RoboDK station: path.rdk

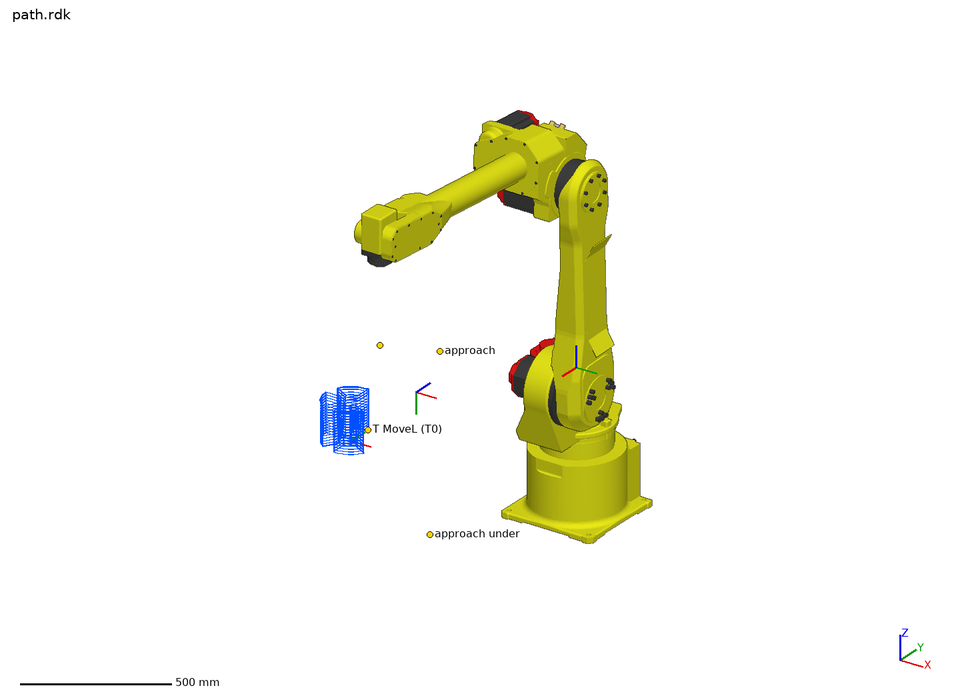
[picture v0: the station drawn from its stored meshes, robots at their saved joint values, targets as dots, program paths as lines]
Station path (saved by RoboDK 5.0.0). Poses are relative to the parent item; angles as X-Y-Z fixed-axis rotations.
  - frame data_frame at (0, 0, 0) mm
    - target approach (Cartesian target) at (94, 380, 204.2) mm, rotated rx -180 ry 0 rz 0 deg; joints [10.247, -49.52, -8.659, -50.211, 13.385, 139.433] of Fanuc ARC Mate 120iB/10L
    - target approach_vert (Cartesian target) at (0, 170, 284.2) mm, rotated rx -90 ry 0 rz 180 deg; joints [0, 2.156, 3.881, -180, 93.881, 90] of Fanuc ARC Mate 120iB/10L
    - target approach under (Cartesian target) at (94, 320, -445.8) mm; joints [3.897, 48.417, -53.03, 175.127, 126.871, 267.072] of Fanuc ARC Mate 120iB/10L
    - target approach_vert_180 (Cartesian target) at (0, 170, 284.2) mm, rotated rx -90 ry 0 rz 0 deg; joints [0, 2.156, 3.881, -180, 93.881, -90] of Fanuc ARC Mate 120iB/10L
    - object path at (0, 0, 0) mm
    - target T MoveL (T0) (Cartesian target) at (0, 100, 0) mm, rotated rx -90 ry 0 rz 0 deg; joints [0, 0, 0, 0, 0, 0] of Fanuc ARC Mate 120iB/10L
  - frame Fanuc ARC Mate 120iB/10L Base at (0, 1300, -250) mm, rotated rx 0 ry 0 rz -90 deg
    - robot Fanuc ARC Mate 120iB/10L: 6 axes, payload 10 kg, reach 1885 mm, repeatability 0.1 mm, weight 225 kg
        modified DH rows (alpha deg, a mm, theta deg, d mm): 0, 0, 0, 525; -90, 150, -90, 0; 0, 770, 0, 0; -90, 100, 0, 960; 90, 0, 0, 0; -90, 0, 0, 100
        base shift (0, 0, -525) mm
        joint limits [-170, -80, -170, -200, -140, -450] to [170, 170, 250, 200, 140, 450]; home [0, 0, 0, 0, 0, 0]; saved at [0, 2.156, 3.881, -180, 93.881, -90]
      - tool Tool 1, TCP at (0, 0, 300) mm, rotated rx 90 ry 0 rz 0 deg
      - tool Tool 2, TCP at (0, 0, 200) mm
      - tool Tool 3, TCP at (0, 0, 300) mm, rotated rx -90 ry 0 rz 0 deg
  - frame Frame 3 at (130, 190, 140) mm, rotated rx -90 ry 0 rz 0 deg
  - program AutoProgram (841 instructions, listed below)
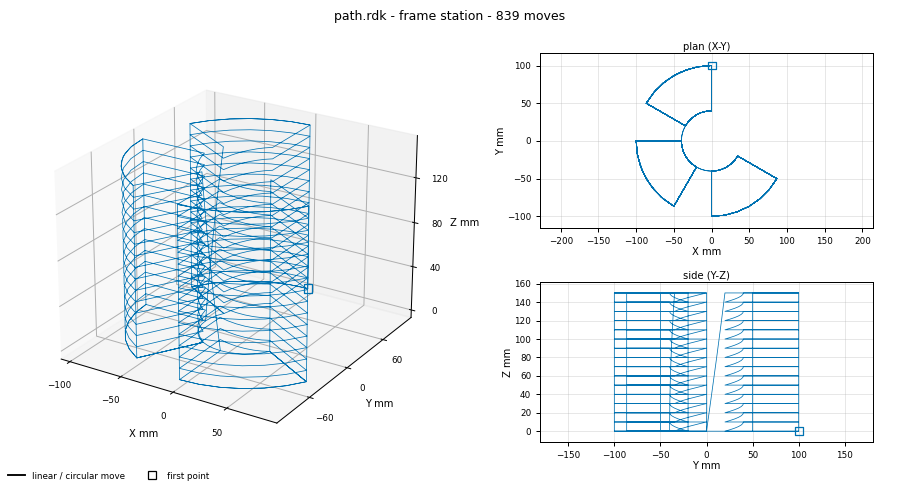
[picture p0: tool path of path.rdk in frame station, 839 of 839 moves have a stored position in this frame; points joined in program order, loops and branches not executed]

--- program AutoProgram (robot Fanuc ARC Mate 120iB/10L) ---
  Set Ref.: data_frame
  Set Tool: Tool 1
  *MoveL (T0) -> target T MoveL (T0)
  MoveL (T1) to (-17.36, 98.48, 0) mm, rotated rx -90 ry 0 rz 10 deg; joints []
  MoveL (T2) to (-34.2, 93.97, 0) mm, rotated rx -90 ry 0 rz 20 deg; joints []
  MoveL (T3) to (-50, 86.6, 0) mm, rotated rx -90 ry 0 rz 30 deg; joints []
  MoveL (T4) to (-64.28, 76.6, 0) mm, rotated rx -90 ry 0 rz 40 deg; joints []
  MoveL (T5) to (-76.6, 64.28, 0) mm, rotated rx -90 ry 0 rz 50 deg; joints []
  MoveL (T6) to (-86.6, 50, 0) mm, rotated rx -90 ry 0 rz 60 deg; joints []
  MoveL (T7) to (-34.64, 20, 0) mm, rotated rx -90 ry 0 rz 60 deg; joints []
  MoveL (T8) to (-30.64, 25.71, 1.67) mm, rotated rx -90 ry 0 rz 50 deg; joints []
  MoveL (T9) to (-25.71, 30.64, 3.33) mm, rotated rx -90 ry 0 rz 40 deg; joints []
  MoveL (T10) to (-20, 34.64, 5) mm, rotated rx -90 ry 0 rz 30 deg; joints []
  MoveL (T11) to (-13.68, 37.59, 6.67) mm, rotated rx -90 ry 0 rz 20 deg; joints []
  MoveL (T12) to (-6.95, 39.39, 8.33) mm, rotated rx -90 ry 0 rz 10 deg; joints []
  MoveL (T13) to (0, 40, 10) mm, rotated rx -90 ry 0 rz 0 deg; joints []
  MoveL (T14) to (0, 100, 10) mm, rotated rx -90 ry 0 rz 0 deg; joints []
  MoveL (T15) to (-17.36, 98.48, 10) mm, rotated rx -90 ry 0 rz 10 deg; joints []
  MoveL (T16) to (-34.2, 93.97, 10) mm, rotated rx -90 ry 0 rz 20 deg; joints []
  MoveL (T17) to (-50, 86.6, 10) mm, rotated rx -90 ry 0 rz 30 deg; joints []
  MoveL (T18) to (-64.28, 76.6, 10) mm, rotated rx -90 ry 0 rz 40 deg; joints []
  MoveL (T19) to (-76.6, 64.28, 10) mm, rotated rx -90 ry 0 rz 50 deg; joints []
  MoveL (T20) to (-86.6, 50, 10) mm, rotated rx -90 ry 0 rz 60 deg; joints []
  MoveL (T21) to (-34.64, 20, 10) mm, rotated rx -90 ry 0 rz 60 deg; joints []
  MoveL (T22) to (-30.64, 25.71, 11.67) mm, rotated rx -90 ry 0 rz 50 deg; joints []
  MoveL (T23) to (-25.71, 30.64, 13.33) mm, rotated rx -90 ry 0 rz 40 deg; joints []
  MoveL (T24) to (-20, 34.64, 15) mm, rotated rx -90 ry 0 rz 30 deg; joints []
  MoveL (T25) to (-13.68, 37.59, 16.67) mm, rotated rx -90 ry 0 rz 20 deg; joints []
  MoveL (T26) to (-6.95, 39.39, 18.33) mm, rotated rx -90 ry 0 rz 10 deg; joints []
  MoveL (T27) to (0, 40, 20) mm, rotated rx -90 ry 0 rz 0 deg; joints []
  MoveL (T28) to (0, 100, 20) mm, rotated rx -90 ry 0 rz 0 deg; joints []
  MoveL (T29) to (-17.36, 98.48, 20) mm, rotated rx -90 ry 0 rz 10 deg; joints []
  MoveL (T30) to (-34.2, 93.97, 20) mm, rotated rx -90 ry 0 rz 20 deg; joints []
  MoveL (T31) to (-50, 86.6, 20) mm, rotated rx -90 ry 0 rz 30 deg; joints []
  MoveL (T32) to (-64.28, 76.6, 20) mm, rotated rx -90 ry 0 rz 40 deg; joints []
  MoveL (T33) to (-76.6, 64.28, 20) mm, rotated rx -90 ry 0 rz 50 deg; joints []
  MoveL (T34) to (-86.6, 50, 20) mm, rotated rx -90 ry 0 rz 60 deg; joints []
  MoveL (T35) to (-34.64, 20, 20) mm, rotated rx -90 ry 0 rz 60 deg; joints []
  MoveL (T36) to (-30.64, 25.71, 21.67) mm, rotated rx -90 ry 0 rz 50 deg; joints []
  MoveL (T37) to (-25.71, 30.64, 23.33) mm, rotated rx -90 ry 0 rz 40 deg; joints []
  MoveL (T38) to (-20, 34.64, 25) mm, rotated rx -90 ry 0 rz 30 deg; joints []
  MoveL (T39) to (-13.68, 37.59, 26.67) mm, rotated rx -90 ry 0 rz 20 deg; joints []
  MoveL (T40) to (-6.95, 39.39, 28.33) mm, rotated rx -90 ry 0 rz 10 deg; joints []
  MoveL (T41) to (0, 40, 30) mm, rotated rx -90 ry 0 rz 0 deg; joints []
  MoveL (T42) to (0, 100, 30) mm, rotated rx -90 ry 0 rz 0 deg; joints []
  MoveL (T43) to (-20.79, 97.81, 30) mm, rotated rx -90 ry 0 rz 12 deg; joints []
  MoveL (T44) to (-40.67, 91.36, 30) mm, rotated rx -90 ry 0 rz 24 deg; joints []
  MoveL (T45) to (-58.78, 80.9, 30) mm, rotated rx -90 ry 0 rz 36 deg; joints []
  MoveL (T46) to (-74.31, 66.91, 30) mm, rotated rx -90 ry 0 rz 48 deg; joints []
  MoveL (T47) to (-86.6, 50, 30) mm, rotated rx -90 ry 0 rz 60 deg; joints []
  MoveL (T48) to (-34.64, 20, 30) mm, rotated rx -90 ry 0 rz 60 deg; joints []
  MoveL (T49) to (-30.64, 25.71, 31.67) mm, rotated rx -90 ry 0 rz 50 deg; joints []
  MoveL (T50) to (-25.71, 30.64, 33.33) mm, rotated rx -90 ry 0 rz 40 deg; joints []
  MoveL (T51) to (-20, 34.64, 35) mm, rotated rx -90 ry 0 rz 30 deg; joints []
  MoveL (T52) to (-13.68, 37.59, 36.67) mm, rotated rx -90 ry 0 rz 20 deg; joints []
  MoveL (T53) to (-6.95, 39.39, 38.33) mm, rotated rx -90 ry 0 rz 10 deg; joints []
  MoveL (T54) to (0, 40, 40) mm, rotated rx -90 ry 0 rz 0 deg; joints []
  MoveL (T55) to (0, 100, 40) mm, rotated rx -90 ry 0 rz 0 deg; joints []
  MoveL (T56) to (-17.36, 98.48, 40) mm, rotated rx -90 ry 0 rz 10 deg; joints []
  MoveL (T57) to (-34.2, 93.97, 40) mm, rotated rx -90 ry 0 rz 20 deg; joints []
  MoveL (T58) to (-50, 86.6, 40) mm, rotated rx -90 ry 0 rz 30 deg; joints []
  MoveL (T59) to (-64.28, 76.6, 40) mm, rotated rx -90 ry 0 rz 40 deg; joints []
  MoveL (T60) to (-76.6, 64.28, 40) mm, rotated rx -90 ry 0 rz 50 deg; joints []
  MoveL (T61) to (-86.6, 50, 40) mm, rotated rx -90 ry 0 rz 60 deg; joints []
  MoveL (T62) to (-34.64, 20, 40) mm, rotated rx -90 ry 0 rz 60 deg; joints []
  MoveL (T63) to (-30.64, 25.71, 41.67) mm, rotated rx -90 ry 0 rz 50 deg; joints []
  MoveL (T64) to (-25.71, 30.64, 43.33) mm, rotated rx -90 ry 0 rz 40 deg; joints []
  MoveL (T65) to (-20, 34.64, 45) mm, rotated rx -90 ry 0 rz 30 deg; joints []
  MoveL (T66) to (-13.68, 37.59, 46.67) mm, rotated rx -90 ry 0 rz 20 deg; joints []
  MoveL (T67) to (-6.95, 39.39, 48.33) mm, rotated rx -90 ry 0 rz 10 deg; joints []
  MoveL (T68) to (0, 40, 50) mm, rotated rx -90 ry 0 rz 0 deg; joints []
  MoveL (T69) to (0, 100, 50) mm, rotated rx -90 ry 0 rz 0 deg; joints []
  MoveL (T70) to (-17.36, 98.48, 50) mm, rotated rx -90 ry 0 rz 10 deg; joints []
  MoveL (T71) to (-34.2, 93.97, 50) mm, rotated rx -90 ry 0 rz 20 deg; joints []
  MoveL (T72) to (-50, 86.6, 50) mm, rotated rx -90 ry 0 rz 30 deg; joints []
  MoveL (T73) to (-64.28, 76.6, 50) mm, rotated rx -90 ry 0 rz 40 deg; joints []
  MoveL (T74) to (-76.6, 64.28, 50) mm, rotated rx -90 ry 0 rz 50 deg; joints []
  MoveL (T75) to (-86.6, 50, 50) mm, rotated rx -90 ry 0 rz 60 deg; joints []
  MoveL (T76) to (-34.64, 20, 50) mm, rotated rx -90 ry 0 rz 60 deg; joints []
  MoveL (T77) to (-30.64, 25.71, 51.67) mm, rotated rx -90 ry 0 rz 50 deg; joints []
  MoveL (T78) to (-25.71, 30.64, 53.33) mm, rotated rx -90 ry 0 rz 40 deg; joints []
  MoveL (T79) to (-20, 34.64, 55) mm, rotated rx -90 ry 0 rz 30 deg; joints []
  MoveL (T80) to (-13.68, 37.59, 56.67) mm, rotated rx -90 ry 0 rz 20 deg; joints []
  MoveL (T81) to (-6.95, 39.39, 58.33) mm, rotated rx -90 ry 0 rz 10 deg; joints []
  MoveL (T82) to (0, 40, 60) mm, rotated rx -90 ry 0 rz 0 deg; joints []
  MoveL (T83) to (0, 100, 60) mm, rotated rx -90 ry 0 rz 0 deg; joints []
  MoveL (T84) to (-17.36, 98.48, 60) mm, rotated rx -90 ry 0 rz 10 deg; joints []
  MoveL (T85) to (-34.2, 93.97, 60) mm, rotated rx -90 ry 0 rz 20 deg; joints []
  MoveL (T86) to (-50, 86.6, 60) mm, rotated rx -90 ry 0 rz 30 deg; joints []
  MoveL (T87) to (-64.28, 76.6, 60) mm, rotated rx -90 ry 0 rz 40 deg; joints []
  MoveL (T88) to (-76.6, 64.28, 60) mm, rotated rx -90 ry 0 rz 50 deg; joints []
  MoveL (T89) to (-86.6, 50, 60) mm, rotated rx -90 ry 0 rz 60 deg; joints []
  MoveL (T90) to (-34.64, 20, 60) mm, rotated rx -90 ry 0 rz 60 deg; joints []
  MoveL (T91) to (-30.64, 25.71, 61.67) mm, rotated rx -90 ry 0 rz 50 deg; joints []
  MoveL (T92) to (-25.71, 30.64, 63.33) mm, rotated rx -90 ry 0 rz 40 deg; joints []
  MoveL (T93) to (-20, 34.64, 65) mm, rotated rx -90 ry 0 rz 30 deg; joints []
  MoveL (T94) to (-13.68, 37.59, 66.67) mm, rotated rx -90 ry 0 rz 20 deg; joints []
  MoveL (T95) to (-6.95, 39.39, 68.33) mm, rotated rx -90 ry 0 rz 10 deg; joints []
  MoveL (T96) to (0, 40, 70) mm, rotated rx -90 ry 0 rz 0 deg; joints []
  MoveL (T97) to (0, 100, 70) mm, rotated rx -90 ry 0 rz 0 deg; joints []
  MoveL (T98) to (-17.36, 98.48, 70) mm, rotated rx -90 ry 0 rz 10 deg; joints []
  MoveL (T99) to (-34.2, 93.97, 70) mm, rotated rx -90 ry 0 rz 20 deg; joints []
  MoveL (T100) to (-50, 86.6, 70) mm, rotated rx -90 ry 0 rz 30 deg; joints []
  MoveL (T101) to (-64.28, 76.6, 70) mm, rotated rx -90 ry 0 rz 40 deg; joints []
  MoveL (T102) to (-76.6, 64.28, 70) mm, rotated rx -90 ry 0 rz 50 deg; joints []
  MoveL (T103) to (-86.6, 50, 70) mm, rotated rx -90 ry 0 rz 60 deg; joints []
  MoveL (T104) to (-34.64, 20, 70) mm, rotated rx -90 ry 0 rz 60 deg; joints []
  MoveL (T105) to (-30.64, 25.71, 71.67) mm, rotated rx -90 ry 0 rz 50 deg; joints []
  MoveL (T106) to (-25.71, 30.64, 73.33) mm, rotated rx -90 ry 0 rz 40 deg; joints []
  MoveL (T107) to (-20, 34.64, 75) mm, rotated rx -90 ry 0 rz 30 deg; joints []
  MoveL (T108) to (-13.68, 37.59, 76.67) mm, rotated rx -90 ry 0 rz 20 deg; joints []
  MoveL (T109) to (-6.95, 39.39, 78.33) mm, rotated rx -90 ry 0 rz 10 deg; joints []
  MoveL (T110) to (0, 40, 80) mm, rotated rx -90 ry 0 rz 0 deg; joints []
  MoveL (T111) to (0, 100, 80) mm, rotated rx -90 ry 0 rz 0 deg; joints []
  MoveL (T112) to (-20.79, 97.81, 80) mm, rotated rx -90 ry 0 rz 12 deg; joints []
  MoveL (T113) to (-40.67, 91.36, 80) mm, rotated rx -90 ry 0 rz 24 deg; joints []
  MoveL (T114) to (-58.78, 80.9, 80) mm, rotated rx -90 ry 0 rz 36 deg; joints []
  MoveL (T115) to (-74.31, 66.91, 80) mm, rotated rx -90 ry 0 rz 48 deg; joints []
  MoveL (T116) to (-86.6, 50, 80) mm, rotated rx -90 ry 0 rz 60 deg; joints []
  MoveL (T117) to (-34.64, 20, 80) mm, rotated rx -90 ry 0 rz 60 deg; joints []
  MoveL (T118) to (-30.64, 25.71, 81.67) mm, rotated rx -90 ry 0 rz 50 deg; joints []
  MoveL (T119) to (-25.71, 30.64, 83.33) mm, rotated rx -90 ry 0 rz 40 deg; joints []
  MoveL (T120) to (-20, 34.64, 85) mm, rotated rx -90 ry 0 rz 30 deg; joints []
  MoveL (T121) to (-13.68, 37.59, 86.67) mm, rotated rx -90 ry 0 rz 20 deg; joints []
  MoveL (T122) to (-6.95, 39.39, 88.33) mm, rotated rx -90 ry 0 rz 10 deg; joints []
  MoveL (T123) to (0, 40, 90) mm, rotated rx -90 ry 0 rz 0 deg; joints []
  MoveL (T124) to (0, 100, 90) mm, rotated rx -90 ry 0 rz 0 deg; joints []
  MoveL (T125) to (-20.79, 97.81, 90) mm, rotated rx -90 ry 0 rz 12 deg; joints []
  MoveL (T126) to (-40.67, 91.36, 90) mm, rotated rx -90 ry 0 rz 24 deg; joints []
  MoveL (T127) to (-58.78, 80.9, 90) mm, rotated rx -90 ry 0 rz 36 deg; joints []
  MoveL (T128) to (-74.31, 66.91, 90) mm, rotated rx -90 ry 0 rz 48 deg; joints []
  MoveL (T129) to (-86.6, 50, 90) mm, rotated rx -90 ry 0 rz 60 deg; joints []
  MoveL (T130) to (-34.64, 20, 90) mm, rotated rx -90 ry 0 rz 60 deg; joints []
  MoveL (T131) to (-30.64, 25.71, 91.67) mm, rotated rx -90 ry 0 rz 50 deg; joints []
  MoveL (T132) to (-25.71, 30.64, 93.33) mm, rotated rx -90 ry 0 rz 40 deg; joints []
  MoveL (T133) to (-20, 34.64, 95) mm, rotated rx -90 ry 0 rz 30 deg; joints []
  MoveL (T134) to (-13.68, 37.59, 96.67) mm, rotated rx -90 ry 0 rz 20 deg; joints []
  MoveL (T135) to (-6.95, 39.39, 98.33) mm, rotated rx -90 ry 0 rz 10 deg; joints []
  MoveL (T136) to (0, 40, 100) mm, rotated rx -90 ry 0 rz 0 deg; joints []
  MoveL (T137) to (0, 100, 100) mm, rotated rx -90 ry 0 rz 0 deg; joints []
  MoveL (T138) to (-20.79, 97.81, 100) mm, rotated rx -90 ry 0 rz 12 deg; joints []
  MoveL (T139) to (-40.67, 91.36, 100) mm, rotated rx -90 ry 0 rz 24 deg; joints []
  MoveL (T140) to (-58.78, 80.9, 100) mm, rotated rx -90 ry 0 rz 36 deg; joints []
  MoveL (T141) to (-74.31, 66.91, 100) mm, rotated rx -90 ry 0 rz 48 deg; joints []
  MoveL (T142) to (-86.6, 50, 100) mm, rotated rx -90 ry 0 rz 60 deg; joints []
  MoveL (T143) to (-34.64, 20, 100) mm, rotated rx -90 ry 0 rz 60 deg; joints []
  MoveL (T144) to (-30.64, 25.71, 101.67) mm, rotated rx -90 ry 0 rz 50 deg; joints []
  MoveL (T145) to (-25.71, 30.64, 103.33) mm, rotated rx -90 ry 0 rz 40 deg; joints []
  MoveL (T146) to (-20, 34.64, 105) mm, rotated rx -90 ry 0 rz 30 deg; joints []
  MoveL (T147) to (-13.68, 37.59, 106.67) mm, rotated rx -90 ry 0 rz 20 deg; joints []
  MoveL (T148) to (-6.95, 39.39, 108.33) mm, rotated rx -90 ry 0 rz 10 deg; joints []
  MoveL (T149) to (0, 40, 110) mm, rotated rx -90 ry 0 rz 0 deg; joints []
  MoveL (T150) to (0, 100, 110) mm, rotated rx -90 ry 0 rz 0 deg; joints []
  MoveL (T151) to (-17.36, 98.48, 110) mm, rotated rx -90 ry 0 rz 10 deg; joints []
  MoveL (T152) to (-34.2, 93.97, 110) mm, rotated rx -90 ry 0 rz 20 deg; joints []
  MoveL (T153) to (-50, 86.6, 110) mm, rotated rx -90 ry 0 rz 30 deg; joints []
  MoveL (T154) to (-64.28, 76.6, 110) mm, rotated rx -90 ry 0 rz 40 deg; joints []
  MoveL (T155) to (-76.6, 64.28, 110) mm, rotated rx -90 ry 0 rz 50 deg; joints []
  MoveL (T156) to (-86.6, 50, 110) mm, rotated rx -90 ry 0 rz 60 deg; joints []
  MoveL (T157) to (-34.64, 20, 110) mm, rotated rx -90 ry 0 rz 60 deg; joints []
  MoveL (T158) to (-30.64, 25.71, 111.67) mm, rotated rx -90 ry 0 rz 50 deg; joints []
  MoveL (T159) to (-25.71, 30.64, 113.33) mm, rotated rx -90 ry 0 rz 40 deg; joints []
  MoveL (T160) to (-20, 34.64, 115) mm, rotated rx -90 ry 0 rz 30 deg; joints []
  MoveL (T161) to (-13.68, 37.59, 116.67) mm, rotated rx -90 ry 0 rz 20 deg; joints []
  MoveL (T162) to (-6.95, 39.39, 118.33) mm, rotated rx -90 ry 0 rz 10 deg; joints []
  MoveL (T163) to (0, 40, 120) mm, rotated rx -90 ry 0 rz 0 deg; joints []
  MoveL (T164) to (0, 100, 120) mm, rotated rx -90 ry 0 rz 0 deg; joints []
  MoveL (T165) to (-17.36, 98.48, 120) mm, rotated rx -90 ry 0 rz 10 deg; joints []
  MoveL (T166) to (-34.2, 93.97, 120) mm, rotated rx -90 ry 0 rz 20 deg; joints []
  MoveL (T167) to (-50, 86.6, 120) mm, rotated rx -90 ry 0 rz 30 deg; joints []
  MoveL (T168) to (-64.28, 76.6, 120) mm, rotated rx -90 ry 0 rz 40 deg; joints []
  MoveL (T169) to (-76.6, 64.28, 120) mm, rotated rx -90 ry 0 rz 50 deg; joints []
  MoveL (T170) to (-86.6, 50, 120) mm, rotated rx -90 ry 0 rz 60 deg; joints []
  MoveL (T171) to (-34.64, 20, 120) mm, rotated rx -90 ry 0 rz 60 deg; joints []
  MoveL (T172) to (-30.64, 25.71, 121.67) mm, rotated rx -90 ry 0 rz 50 deg; joints []
  MoveL (T173) to (-25.71, 30.64, 123.33) mm, rotated rx -90 ry 0 rz 40 deg; joints []
  MoveL (T174) to (-20, 34.64, 125) mm, rotated rx -90 ry 0 rz 30 deg; joints []
  MoveL (T175) to (-13.68, 37.59, 126.67) mm, rotated rx -90 ry 0 rz 20 deg; joints []
  MoveL (T176) to (-6.95, 39.39, 128.33) mm, rotated rx -90 ry 0 rz 10 deg; joints []
  MoveL (T177) to (0, 40, 130) mm, rotated rx -90 ry 0 rz 0 deg; joints []
  MoveL (T178) to (0, 100, 130) mm, rotated rx -90 ry 0 rz 0 deg; joints []
  MoveL (T179) to (-17.36, 98.48, 130) mm, rotated rx -90 ry 0 rz 10 deg; joints []
  MoveL (T180) to (-34.2, 93.97, 130) mm, rotated rx -90 ry 0 rz 20 deg; joints []
  MoveL (T181) to (-50, 86.6, 130) mm, rotated rx -90 ry 0 rz 30 deg; joints []
  MoveL (T182) to (-64.28, 76.6, 130) mm, rotated rx -90 ry 0 rz 40 deg; joints []
  MoveL (T183) to (-76.6, 64.28, 130) mm, rotated rx -90 ry 0 rz 50 deg; joints []
  MoveL (T184) to (-86.6, 50, 130) mm, rotated rx -90 ry 0 rz 60 deg; joints []
  MoveL (T185) to (-34.64, 20, 130) mm, rotated rx -90 ry 0 rz 60 deg; joints []
  MoveL (T186) to (-30.64, 25.71, 131.67) mm, rotated rx -90 ry 0 rz 50 deg; joints []
  MoveL (T187) to (-25.71, 30.64, 133.33) mm, rotated rx -90 ry 0 rz 40 deg; joints []
  MoveL (T188) to (-20, 34.64, 135) mm, rotated rx -90 ry 0 rz 30 deg; joints []
  MoveL (T189) to (-13.68, 37.59, 136.67) mm, rotated rx -90 ry 0 rz 20 deg; joints []
  MoveL (T190) to (-6.95, 39.39, 138.33) mm, rotated rx -90 ry 0 rz 10 deg; joints []
  MoveL (T191) to (0, 40, 140) mm, rotated rx -90 ry 0 rz 0 deg; joints []
  MoveL (T192) to (0, 100, 140) mm, rotated rx -90 ry 0 rz 0 deg; joints []
  MoveL (T193) to (-17.36, 98.48, 140) mm, rotated rx -90 ry 0 rz 10 deg; joints []
  MoveL (T194) to (-34.2, 93.97, 140) mm, rotated rx -90 ry 0 rz 20 deg; joints []
  MoveL (T195) to (-50, 86.6, 140) mm, rotated rx -90 ry 0 rz 30 deg; joints []
  MoveL (T196) to (-64.28, 76.6, 140) mm, rotated rx -90 ry 0 rz 40 deg; joints []
  MoveL (T197) to (-76.6, 64.28, 140) mm, rotated rx -90 ry 0 rz 50 deg; joints []
  MoveL (T198) to (-86.6, 50, 140) mm, rotated rx -90 ry 0 rz 60 deg; joints []
  MoveL (T199) to (-34.64, 20, 140) mm, rotated rx -90 ry 0 rz 60 deg; joints []
  MoveL (T200) to (-30.64, 25.71, 141.67) mm, rotated rx -90 ry 0 rz 50 deg; joints []
  MoveL (T201) to (-25.71, 30.64, 143.33) mm, rotated rx -90 ry 0 rz 40 deg; joints []
  MoveL (T202) to (-20, 34.64, 145) mm, rotated rx -90 ry 0 rz 30 deg; joints []
  MoveL (T203) to (-13.68, 37.59, 146.67) mm, rotated rx -90 ry 0 rz 20 deg; joints []
  MoveL (T204) to (-6.95, 39.39, 148.33) mm, rotated rx -90 ry 0 rz 10 deg; joints []
  MoveL (T205) to (0, 40, 150) mm, rotated rx -90 ry 0 rz 0 deg; joints []
  MoveL (T206) to (0, 100, 150) mm, rotated rx -90 ry 0 rz 0 deg; joints []
  MoveL (T207) to (-17.36, 98.48, 150) mm, rotated rx -90 ry 0 rz 10 deg; joints []
  MoveL (T208) to (-34.2, 93.97, 150) mm, rotated rx -90 ry 0 rz 20 deg; joints []
  MoveL (T209) to (-50, 86.6, 150) mm, rotated rx -90 ry 0 rz 30 deg; joints []
  MoveL (T210) to (-64.28, 76.6, 150) mm, rotated rx -90 ry 0 rz 40 deg; joints []
  MoveL (T211) to (-76.6, 64.28, 150) mm, rotated rx -90 ry 0 rz 50 deg; joints []
  MoveL (T212) to (-86.6, 50, 150) mm, rotated rx -90 ry 0 rz 60 deg; joints []
  MoveL (T213) to (-34.64, 20, 150) mm, rotated rx -90 ry 0 rz 60 deg; joints []
  MoveL (T214) to (-35.32, 18.78, 140) mm, rotated rx -90 ry 0 rz 62 deg; joints []
  MoveL (T215) to (-35.95, 17.54, 130) mm, rotated rx -90 ry 0 rz 64 deg; joints []
  MoveL (T216) to (-36.54, 16.27, 120) mm, rotated rx -90 ry 0 rz 66 deg; joints []
  MoveL (T217) to (-37.09, 14.98, 110) mm, rotated rx -90 ry 0 rz 68 deg; joints []
  MoveL (T218) to (-37.59, 13.68, 100) mm, rotated rx -90 ry 0 rz 70 deg; joints []
  MoveL (T219) to (-38.04, 12.36, 90) mm, rotated rx -90 ry 0 rz 72 deg; joints []
  MoveL (T220) to (-38.45, 11.03, 80) mm, rotated rx -90 ry 0 rz 74 deg; joints []
  MoveL (T221) to (-38.81, 9.68, 70) mm, rotated rx -90 ry 0 rz 76 deg; joints []
  MoveL (T222) to (-39.13, 8.32, 60) mm, rotated rx -90 ry 0 rz 78 deg; joints []
  MoveL (T223) to (-39.39, 6.95, 50) mm, rotated rx -90 ry 0 rz 80 deg; joints []
  MoveL (T224) to (-39.61, 5.57, 40) mm, rotated rx -90 ry 0 rz 82 deg; joints []
  MoveL (T225) to (-39.78, 4.18, 30) mm, rotated rx -90 ry 0 rz 84 deg; joints []
  MoveL (T226) to (-39.9, 2.79, 20) mm, rotated rx -90 ry 0 rz 86 deg; joints []
  MoveL (T227) to (-39.98, 1.4, 10) mm, rotated rx -90 ry 0 rz 88 deg; joints []
  MoveL (T228) to (-40, 0, 0) mm, rotated rx -90 ry 0 rz 90 deg; joints []
  MoveL (T229) to (-100, 0, 0) mm, rotated rx -90 ry 0 rz 90 deg; joints []
  MoveL (T230) to (-98.48, -17.36, 0) mm, rotated rx -90 ry 0 rz 100 deg; joints []
  MoveL (T231) to (-93.97, -34.2, 0) mm, rotated rx -90 ry 0 rz 110 deg; joints []
  MoveL (T232) to (-86.6, -50, 0) mm, rotated rx -90 ry 0 rz 120 deg; joints []
  MoveL (T233) to (-76.6, -64.28, 0) mm, rotated rx -90 ry 0 rz 130 deg; joints []
  MoveL (T234) to (-64.28, -76.6, 0) mm, rotated rx -90 ry 0 rz 140 deg; joints []
  MoveL (T235) to (-50, -86.6, 0) mm, rotated rx -90 ry 0 rz 150 deg; joints []
  MoveL (T236) to (-20, -34.64, 0) mm, rotated rx -90 ry 0 rz 150 deg; joints []
  MoveL (T237) to (-25.71, -30.64, 1.67) mm, rotated rx -90 ry 0 rz 140 deg; joints []
  MoveL (T238) to (-30.64, -25.71, 3.33) mm, rotated rx -90 ry 0 rz 130 deg; joints []
  MoveL (T239) to (-34.64, -20, 5) mm, rotated rx -90 ry 0 rz 120 deg; joints []
  MoveL (T240) to (-37.59, -13.68, 6.67) mm, rotated rx -90 ry 0 rz 110 deg; joints []
  MoveL (T241) to (-39.39, -6.95, 8.33) mm, rotated rx -90 ry 0 rz 100 deg; joints []
  MoveL (T242) to (-40, 0, 10) mm, rotated rx -90 ry 0 rz 90 deg; joints []
  MoveL (T243) to (-100, 0, 10) mm, rotated rx -90 ry 0 rz 90 deg; joints []
  MoveL (T244) to (-98.48, -17.36, 10) mm, rotated rx -90 ry 0 rz 100 deg; joints []
  MoveL (T245) to (-93.97, -34.2, 10) mm, rotated rx -90 ry 0 rz 110 deg; joints []
  MoveL (T246) to (-86.6, -50, 10) mm, rotated rx -90 ry 0 rz 120 deg; joints []
  MoveL (T247) to (-76.6, -64.28, 10) mm, rotated rx -90 ry 0 rz 130 deg; joints []
  MoveL (T248) to (-64.28, -76.6, 10) mm, rotated rx -90 ry 0 rz 140 deg; joints []
  MoveL (T249) to (-50, -86.6, 10) mm, rotated rx -90 ry 0 rz 150 deg; joints []
  MoveL (T250) to (-20, -34.64, 10) mm, rotated rx -90 ry 0 rz 150 deg; joints []
  MoveL (T251) to (-25.71, -30.64, 11.67) mm, rotated rx -90 ry 0 rz 140 deg; joints []
  MoveL (T252) to (-30.64, -25.71, 13.33) mm, rotated rx -90 ry 0 rz 130 deg; joints []
  MoveL (T253) to (-34.64, -20, 15) mm, rotated rx -90 ry 0 rz 120 deg; joints []
  MoveL (T254) to (-37.59, -13.68, 16.67) mm, rotated rx -90 ry 0 rz 110 deg; joints []
  MoveL (T255) to (-39.39, -6.95, 18.33) mm, rotated rx -90 ry 0 rz 100 deg; joints []
  MoveL (T256) to (-40, 0, 20) mm, rotated rx -90 ry 0 rz 90 deg; joints []
  MoveL (T257) to (-100, 0, 20) mm, rotated rx -90 ry 0 rz 90 deg; joints []
  MoveL (T258) to (-98.48, -17.36, 20) mm, rotated rx -90 ry 0 rz 100 deg; joints []
  MoveL (T259) to (-93.97, -34.2, 20) mm, rotated rx -90 ry 0 rz 110 deg; joints []
  MoveL (T260) to (-86.6, -50, 20) mm, rotated rx -90 ry 0 rz 120 deg; joints []
  MoveL (T261) to (-76.6, -64.28, 20) mm, rotated rx -90 ry 0 rz 130 deg; joints []
  MoveL (T262) to (-64.28, -76.6, 20) mm, rotated rx -90 ry 0 rz 140 deg; joints []
  MoveL (T263) to (-50, -86.6, 20) mm, rotated rx -90 ry 0 rz 150 deg; joints []
  MoveL (T264) to (-20, -34.64, 20) mm, rotated rx -90 ry 0 rz 150 deg; joints []
  MoveL (T265) to (-25.71, -30.64, 21.67) mm, rotated rx -90 ry 0 rz 140 deg; joints []
  MoveL (T266) to (-30.64, -25.71, 23.33) mm, rotated rx -90 ry 0 rz 130 deg; joints []
  MoveL (T267) to (-34.64, -20, 25) mm, rotated rx -90 ry 0 rz 120 deg; joints []
  MoveL (T268) to (-37.59, -13.68, 26.67) mm, rotated rx -90 ry 0 rz 110 deg; joints []
  MoveL (T269) to (-39.39, -6.95, 28.33) mm, rotated rx -90 ry 0 rz 100 deg; joints []
  MoveL (T270) to (-40, 0, 30) mm, rotated rx -90 ry 0 rz 90 deg; joints []
  MoveL (T271) to (-100, 0, 30) mm, rotated rx -90 ry 0 rz 90 deg; joints []
  MoveL (T272) to (-98.48, -17.36, 30) mm, rotated rx -90 ry 0 rz 100 deg; joints []
  MoveL (T273) to (-93.97, -34.2, 30) mm, rotated rx -90 ry 0 rz 110 deg; joints []
  MoveL (T274) to (-86.6, -50, 30) mm, rotated rx -90 ry 0 rz 120 deg; joints []
  MoveL (T275) to (-76.6, -64.28, 30) mm, rotated rx -90 ry 0 rz 130 deg; joints []
  MoveL (T276) to (-64.28, -76.6, 30) mm, rotated rx -90 ry 0 rz 140 deg; joints []
  MoveL (T277) to (-50, -86.6, 30) mm, rotated rx -90 ry 0 rz 150 deg; joints []
  MoveL (T278) to (-20, -34.64, 30) mm, rotated rx -90 ry 0 rz 150 deg; joints []
  MoveL (T279) to (-25.71, -30.64, 31.67) mm, rotated rx -90 ry 0 rz 140 deg; joints []
  MoveL (T280) to (-30.64, -25.71, 33.33) mm, rotated rx -90 ry 0 rz 130 deg; joints []
  MoveL (T281) to (-34.64, -20, 35) mm, rotated rx -90 ry 0 rz 120 deg; joints []
  MoveL (T282) to (-37.59, -13.68, 36.67) mm, rotated rx -90 ry 0 rz 110 deg; joints []
  MoveL (T283) to (-39.39, -6.95, 38.33) mm, rotated rx -90 ry 0 rz 100 deg; joints []
  MoveL (T284) to (-40, 0, 40) mm, rotated rx -90 ry 0 rz 90 deg; joints []
  MoveL (T285) to (-100, 0, 40) mm, rotated rx -90 ry 0 rz 90 deg; joints []
  MoveL (T286) to (-98.48, -17.36, 40) mm, rotated rx -90 ry 0 rz 100 deg; joints []
  MoveL (T287) to (-93.97, -34.2, 40) mm, rotated rx -90 ry 0 rz 110 deg; joints []
  MoveL (T288) to (-86.6, -50, 40) mm, rotated rx -90 ry 0 rz 120 deg; joints []
  MoveL (T289) to (-76.6, -64.28, 40) mm, rotated rx -90 ry 0 rz 130 deg; joints []
  MoveL (T290) to (-64.28, -76.6, 40) mm, rotated rx -90 ry 0 rz 140 deg; joints []
  MoveL (T291) to (-50, -86.6, 40) mm, rotated rx -90 ry 0 rz 150 deg; joints []
  MoveL (T292) to (-20, -34.64, 40) mm, rotated rx -90 ry 0 rz 150 deg; joints []
  MoveL (T293) to (-25.71, -30.64, 41.67) mm, rotated rx -90 ry 0 rz 140 deg; joints []
  MoveL (T294) to (-30.64, -25.71, 43.33) mm, rotated rx -90 ry 0 rz 130 deg; joints []
  MoveL (T295) to (-34.64, -20, 45) mm, rotated rx -90 ry 0 rz 120 deg; joints []
  MoveL (T296) to (-37.59, -13.68, 46.67) mm, rotated rx -90 ry 0 rz 110 deg; joints []
  MoveL (T297) to (-39.39, -6.95, 48.33) mm, rotated rx -90 ry 0 rz 100 deg; joints []
  MoveL (T298) to (-40, 0, 50) mm, rotated rx -90 ry 0 rz 90 deg; joints []
  MoveL (T299) to (-100, 0, 50) mm, rotated rx -90 ry 0 rz 90 deg; joints []
  MoveL (T300) to (-98.48, -17.36, 50) mm, rotated rx -90 ry 0 rz 100 deg; joints []
  MoveL (T301) to (-93.97, -34.2, 50) mm, rotated rx -90 ry 0 rz 110 deg; joints []
  MoveL (T302) to (-86.6, -50, 50) mm, rotated rx -90 ry 0 rz 120 deg; joints []
  MoveL (T303) to (-76.6, -64.28, 50) mm, rotated rx -90 ry 0 rz 130 deg; joints []
  MoveL (T304) to (-64.28, -76.6, 50) mm, rotated rx -90 ry 0 rz 140 deg; joints []
  MoveL (T305) to (-50, -86.6, 50) mm, rotated rx -90 ry 0 rz 150 deg; joints []
  MoveL (T306) to (-20, -34.64, 50) mm, rotated rx -90 ry 0 rz 150 deg; joints []
  MoveL (T307) to (-25.71, -30.64, 51.67) mm, rotated rx -90 ry 0 rz 140 deg; joints []
  MoveL (T308) to (-30.64, -25.71, 53.33) mm, rotated rx -90 ry 0 rz 130 deg; joints []
  MoveL (T309) to (-34.64, -20, 55) mm, rotated rx -90 ry 0 rz 120 deg; joints []
  MoveL (T310) to (-37.59, -13.68, 56.67) mm, rotated rx -90 ry 0 rz 110 deg; joints []
  MoveL (T311) to (-39.39, -6.95, 58.33) mm, rotated rx -90 ry 0 rz 100 deg; joints []
  MoveL (T312) to (-40, 0, 60) mm, rotated rx -90 ry 0 rz 90 deg; joints []
  MoveL (T313) to (-100, 0, 60) mm, rotated rx -90 ry 0 rz 90 deg; joints []
  MoveL (T314) to (-98.48, -17.36, 60) mm, rotated rx -90 ry 0 rz 100 deg; joints []
  MoveL (T315) to (-93.97, -34.2, 60) mm, rotated rx -90 ry 0 rz 110 deg; joints []
  MoveL (T316) to (-86.6, -50, 60) mm, rotated rx -90 ry 0 rz 120 deg; joints []
  MoveL (T317) to (-76.6, -64.28, 60) mm, rotated rx -90 ry 0 rz 130 deg; joints []
  MoveL (T318) to (-64.28, -76.6, 60) mm, rotated rx -90 ry 0 rz 140 deg; joints []
  MoveL (T319) to (-50, -86.6, 60) mm, rotated rx -90 ry 0 rz 150 deg; joints []
  MoveL (T320) to (-20, -34.64, 60) mm, rotated rx -90 ry 0 rz 150 deg; joints []
  MoveL (T321) to (-25.71, -30.64, 61.67) mm, rotated rx -90 ry 0 rz 140 deg; joints []
  MoveL (T322) to (-30.64, -25.71, 63.33) mm, rotated rx -90 ry 0 rz 130 deg; joints []
  MoveL (T323) to (-34.64, -20, 65) mm, rotated rx -90 ry 0 rz 120 deg; joints []
  MoveL (T324) to (-37.59, -13.68, 66.67) mm, rotated rx -90 ry 0 rz 110 deg; joints []
  MoveL (T325) to (-39.39, -6.95, 68.33) mm, rotated rx -90 ry 0 rz 100 deg; joints []
  MoveL (T326) to (-40, 0, 70) mm, rotated rx -90 ry 0 rz 90 deg; joints []
  MoveL (T327) to (-100, 0, 70) mm, rotated rx -90 ry 0 rz 90 deg; joints []
  MoveL (T328) to (-98.48, -17.36, 70) mm, rotated rx -90 ry 0 rz 100 deg; joints []
  MoveL (T329) to (-93.97, -34.2, 70) mm, rotated rx -90 ry 0 rz 110 deg; joints []
  MoveL (T330) to (-86.6, -50, 70) mm, rotated rx -90 ry 0 rz 120 deg; joints []
  MoveL (T331) to (-76.6, -64.28, 70) mm, rotated rx -90 ry 0 rz 130 deg; joints []
  MoveL (T332) to (-64.28, -76.6, 70) mm, rotated rx -90 ry 0 rz 140 deg; joints []
  MoveL (T333) to (-50, -86.6, 70) mm, rotated rx -90 ry 0 rz 150 deg; joints []
  MoveL (T334) to (-20, -34.64, 70) mm, rotated rx -90 ry 0 rz 150 deg; joints []
  MoveL (T335) to (-25.71, -30.64, 71.67) mm, rotated rx -90 ry 0 rz 140 deg; joints []
  MoveL (T336) to (-30.64, -25.71, 73.33) mm, rotated rx -90 ry 0 rz 130 deg; joints []
  MoveL (T337) to (-34.64, -20, 75) mm, rotated rx -90 ry 0 rz 120 deg; joints []
  MoveL (T338) to (-37.59, -13.68, 76.67) mm, rotated rx -90 ry 0 rz 110 deg; joints []
  MoveL (T339) to (-39.39, -6.95, 78.33) mm, rotated rx -90 ry 0 rz 100 deg; joints []
  MoveL (T340) to (-40, 0, 80) mm, rotated rx -90 ry 0 rz 90 deg; joints []
  MoveL (T341) to (-100, 0, 80) mm, rotated rx -90 ry 0 rz 90 deg; joints []
  MoveL (T342) to (-98.48, -17.36, 80) mm, rotated rx -90 ry 0 rz 100 deg; joints []
  MoveL (T343) to (-93.97, -34.2, 80) mm, rotated rx -90 ry 0 rz 110 deg; joints []
  MoveL (T344) to (-86.6, -50, 80) mm, rotated rx -90 ry 0 rz 120 deg; joints []
  MoveL (T345) to (-76.6, -64.28, 80) mm, rotated rx -90 ry 0 rz 130 deg; joints []
  MoveL (T346) to (-64.28, -76.6, 80) mm, rotated rx -90 ry 0 rz 140 deg; joints []
  MoveL (T347) to (-50, -86.6, 80) mm, rotated rx -90 ry 0 rz 150 deg; joints []
  MoveL (T348) to (-20, -34.64, 80) mm, rotated rx -90 ry 0 rz 150 deg; joints []
  MoveL (T349) to (-25.71, -30.64, 81.67) mm, rotated rx -90 ry 0 rz 140 deg; joints []
  MoveL (T350) to (-30.64, -25.71, 83.33) mm, rotated rx -90 ry 0 rz 130 deg; joints []
  MoveL (T351) to (-34.64, -20, 85) mm, rotated rx -90 ry 0 rz 120 deg; joints []
  MoveL (T352) to (-37.59, -13.68, 86.67) mm, rotated rx -90 ry 0 rz 110 deg; joints []
  MoveL (T353) to (-39.39, -6.95, 88.33) mm, rotated rx -90 ry 0 rz 100 deg; joints []
  MoveL (T354) to (-40, 0, 90) mm, rotated rx -90 ry 0 rz 90 deg; joints []
  MoveL (T355) to (-100, 0, 90) mm, rotated rx -90 ry 0 rz 90 deg; joints []
  MoveL (T356) to (-98.48, -17.36, 90) mm, rotated rx -90 ry 0 rz 100 deg; joints []
  MoveL (T357) to (-93.97, -34.2, 90) mm, rotated rx -90 ry 0 rz 110 deg; joints []
  MoveL (T358) to (-86.6, -50, 90) mm, rotated rx -90 ry 0 rz 120 deg; joints []
  MoveL (T359) to (-76.6, -64.28, 90) mm, rotated rx -90 ry 0 rz 130 deg; joints []
  MoveL (T360) to (-64.28, -76.6, 90) mm, rotated rx -90 ry 0 rz 140 deg; joints []
  MoveL (T361) to (-50, -86.6, 90) mm, rotated rx -90 ry 0 rz 150 deg; joints []
  MoveL (T362) to (-20, -34.64, 90) mm, rotated rx -90 ry 0 rz 150 deg; joints []
  MoveL (T363) to (-25.71, -30.64, 91.67) mm, rotated rx -90 ry 0 rz 140 deg; joints []
  MoveL (T364) to (-30.64, -25.71, 93.33) mm, rotated rx -90 ry 0 rz 130 deg; joints []
  MoveL (T365) to (-34.64, -20, 95) mm, rotated rx -90 ry 0 rz 120 deg; joints []
  MoveL (T366) to (-37.59, -13.68, 96.67) mm, rotated rx -90 ry 0 rz 110 deg; joints []
  MoveL (T367) to (-39.39, -6.95, 98.33) mm, rotated rx -90 ry 0 rz 100 deg; joints []
  MoveL (T368) to (-40, 0, 100) mm, rotated rx -90 ry 0 rz 90 deg; joints []
  MoveL (T369) to (-100, 0, 100) mm, rotated rx -90 ry 0 rz 90 deg; joints []
  MoveL (T370) to (-98.48, -17.36, 100) mm, rotated rx -90 ry 0 rz 100 deg; joints []
  MoveL (T371) to (-93.97, -34.2, 100) mm, rotated rx -90 ry 0 rz 110 deg; joints []
  MoveL (T372) to (-86.6, -50, 100) mm, rotated rx -90 ry 0 rz 120 deg; joints []
  MoveL (T373) to (-76.6, -64.28, 100) mm, rotated rx -90 ry 0 rz 130 deg; joints []
  MoveL (T374) to (-64.28, -76.6, 100) mm, rotated rx -90 ry 0 rz 140 deg; joints []
  MoveL (T375) to (-50, -86.6, 100) mm, rotated rx -90 ry 0 rz 150 deg; joints []
  MoveL (T376) to (-20, -34.64, 100) mm, rotated rx -90 ry 0 rz 150 deg; joints []
  MoveL (T377) to (-25.71, -30.64, 101.67) mm, rotated rx -90 ry 0 rz 140 deg; joints []
  MoveL (T378) to (-30.64, -25.71, 103.33) mm, rotated rx -90 ry 0 rz 130 deg; joints []
  MoveL (T379) to (-34.64, -20, 105) mm, rotated rx -90 ry 0 rz 120 deg; joints []
  MoveL (T380) to (-37.59, -13.68, 106.67) mm, rotated rx -90 ry 0 rz 110 deg; joints []
  MoveL (T381) to (-39.39, -6.95, 108.33) mm, rotated rx -90 ry 0 rz 100 deg; joints []
  MoveL (T382) to (-40, 0, 110) mm, rotated rx -90 ry 0 rz 90 deg; joints []
  MoveL (T383) to (-100, 0, 110) mm, rotated rx -90 ry 0 rz 90 deg; joints []
  MoveL (T384) to (-97.81, -20.79, 110) mm, rotated rx -90 ry 0 rz 102 deg; joints []
  MoveL (T385) to (-91.36, -40.67, 110) mm, rotated rx -90 ry 0 rz 114 deg; joints []
  MoveL (T386) to (-80.9, -58.78, 110) mm, rotated rx -90 ry 0 rz 126 deg; joints []
  MoveL (T387) to (-66.91, -74.31, 110) mm, rotated rx -90 ry 0 rz 138 deg; joints []
  MoveL (T388) to (-50, -86.6, 110) mm, rotated rx -90 ry 0 rz 150 deg; joints []
  MoveL (T389) to (-20, -34.64, 110) mm, rotated rx -90 ry 0 rz 150 deg; joints []
  MoveL (T390) to (-25.71, -30.64, 111.67) mm, rotated rx -90 ry 0 rz 140 deg; joints []
  MoveL (T391) to (-30.64, -25.71, 113.33) mm, rotated rx -90 ry 0 rz 130 deg; joints []
  MoveL (T392) to (-34.64, -20, 115) mm, rotated rx -90 ry 0 rz 120 deg; joints []
  MoveL (T393) to (-37.59, -13.68, 116.67) mm, rotated rx -90 ry 0 rz 110 deg; joints []
  MoveL (T394) to (-39.39, -6.95, 118.33) mm, rotated rx -90 ry 0 rz 100 deg; joints []
  MoveL (T395) to (-40, 0, 120) mm, rotated rx -90 ry 0 rz 90 deg; joints []
  MoveL (T396) to (-100, 0, 120) mm, rotated rx -90 ry 0 rz 90 deg; joints []
  MoveL (T397) to (-97.81, -20.79, 120) mm, rotated rx -90 ry 0 rz 102 deg; joints []
  MoveL (T398) to (-91.36, -40.67, 120) mm, rotated rx -90 ry 0 rz 114 deg; joints []
  MoveL (T399) to (-80.9, -58.78, 120) mm, rotated rx -90 ry 0 rz 126 deg; joints []
  MoveL (T400) to (-66.91, -74.31, 120) mm, rotated rx -90 ry 0 rz 138 deg; joints []
  MoveL (T401) to (-50, -86.6, 120) mm, rotated rx -90 ry 0 rz 150 deg; joints []
  MoveL (T402) to (-20, -34.64, 120) mm, rotated rx -90 ry 0 rz 150 deg; joints []
  MoveL (T403) to (-25.71, -30.64, 121.67) mm, rotated rx -90 ry 0 rz 140 deg; joints []
  MoveL (T404) to (-30.64, -25.71, 123.33) mm, rotated rx -90 ry 0 rz 130 deg; joints []
  MoveL (T405) to (-34.64, -20, 125) mm, rotated rx -90 ry 0 rz 120 deg; joints []
  MoveL (T406) to (-37.59, -13.68, 126.67) mm, rotated rx -90 ry 0 rz 110 deg; joints []
  MoveL (T407) to (-39.39, -6.95, 128.33) mm, rotated rx -90 ry 0 rz 100 deg; joints []
  MoveL (T408) to (-40, 0, 130) mm, rotated rx -90 ry 0 rz 90 deg; joints []
  MoveL (T409) to (-100, 0, 130) mm, rotated rx -90 ry 0 rz 90 deg; joints []
  MoveL (T410) to (-97.81, -20.79, 130) mm, rotated rx -90 ry 0 rz 102 deg; joints []
  MoveL (T411) to (-91.36, -40.67, 130) mm, rotated rx -90 ry 0 rz 114 deg; joints []
  MoveL (T412) to (-80.9, -58.78, 130) mm, rotated rx -90 ry 0 rz 126 deg; joints []
  MoveL (T413) to (-66.91, -74.31, 130) mm, rotated rx -90 ry 0 rz 138 deg; joints []
  MoveL (T414) to (-50, -86.6, 130) mm, rotated rx -90 ry 0 rz 150 deg; joints []
  MoveL (T415) to (-20, -34.64, 130) mm, rotated rx -90 ry 0 rz 150 deg; joints []
  MoveL (T416) to (-25.71, -30.64, 131.67) mm, rotated rx -90 ry 0 rz 140 deg; joints []
  MoveL (T417) to (-30.64, -25.71, 133.33) mm, rotated rx -90 ry 0 rz 130 deg; joints []
  MoveL (T418) to (-34.64, -20, 135) mm, rotated rx -90 ry 0 rz 120 deg; joints []
  MoveL (T419) to (-37.59, -13.68, 136.67) mm, rotated rx -90 ry 0 rz 110 deg; joints []
  MoveL (T420) to (-39.39, -6.95, 138.33) mm, rotated rx -90 ry 0 rz 100 deg; joints []
  MoveL (T421) to (-40, 0, 140) mm, rotated rx -90 ry 0 rz 90 deg; joints []
  MoveL (T422) to (-100, 0, 140) mm, rotated rx -90 ry 0 rz 90 deg; joints []
  MoveL (T423) to (-97.81, -20.79, 140) mm, rotated rx -90 ry 0 rz 102 deg; joints []
  MoveL (T424) to (-91.36, -40.67, 140) mm, rotated rx -90 ry 0 rz 114 deg; joints []
  MoveL (T425) to (-80.9, -58.78, 140) mm, rotated rx -90 ry 0 rz 126 deg; joints []
  MoveL (T426) to (-66.91, -74.31, 140) mm, rotated rx -90 ry 0 rz 138 deg; joints []
  MoveL (T427) to (-50, -86.6, 140) mm, rotated rx -90 ry 0 rz 150 deg; joints []
  MoveL (T428) to (-20, -34.64, 140) mm, rotated rx -90 ry 0 rz 150 deg; joints []
  MoveL (T429) to (-25.71, -30.64, 141.67) mm, rotated rx -90 ry 0 rz 140 deg; joints []
  MoveL (T430) to (-30.64, -25.71, 143.33) mm, rotated rx -90 ry 0 rz 130 deg; joints []
  MoveL (T431) to (-34.64, -20, 145) mm, rotated rx -90 ry 0 rz 120 deg; joints []
  MoveL (T432) to (-37.59, -13.68, 146.67) mm, rotated rx -90 ry 0 rz 110 deg; joints []
  MoveL (T433) to (-39.39, -6.95, 148.33) mm, rotated rx -90 ry 0 rz 100 deg; joints []
  MoveL (T434) to (-40, 0, 150) mm, rotated rx -90 ry 0 rz 90 deg; joints []
  MoveL (T435) to (-100, 0, 150) mm, rotated rx -90 ry 0 rz 90 deg; joints []
  MoveL (T436) to (-97.81, -20.79, 150) mm, rotated rx -90 ry 0 rz 102 deg; joints []
  MoveL (T437) to (-91.36, -40.67, 150) mm, rotated rx -90 ry 0 rz 114 deg; joints []
  MoveL (T438) to (-80.9, -58.78, 150) mm, rotated rx -90 ry 0 rz 126 deg; joints []
  MoveL (T439) to (-66.91, -74.31, 150) mm, rotated rx -90 ry 0 rz 138 deg; joints []
  MoveL (T440) to (-50, -86.6, 150) mm, rotated rx -90 ry 0 rz 150 deg; joints []
  MoveL (T441) to (-20, -34.64, 150) mm, rotated rx -90 ry 0 rz 150 deg; joints []
  MoveL (T442) to (-18.78, -35.32, 140) mm, rotated rx -90 ry 0 rz 152 deg; joints []
  MoveL (T443) to (-17.54, -35.95, 130) mm, rotated rx -90 ry 0 rz 154 deg; joints []
  MoveL (T444) to (-16.27, -36.54, 120) mm, rotated rx -90 ry 0 rz 156 deg; joints []
  MoveL (T445) to (-14.98, -37.09, 110) mm, rotated rx -90 ry 0 rz 158 deg; joints []
  MoveL (T446) to (-13.68, -37.59, 100) mm, rotated rx -90 ry 0 rz 160 deg; joints []
  MoveL (T447) to (-12.36, -38.04, 90) mm, rotated rx -90 ry 0 rz 162 deg; joints []
  MoveL (T448) to (-11.03, -38.45, 80) mm, rotated rx -90 ry 0 rz 164 deg; joints []
  MoveL (T449) to (-9.68, -38.81, 70) mm, rotated rx -90 ry 0 rz 166 deg; joints []
  MoveL (T450) to (-8.32, -39.13, 60) mm, rotated rx -90 ry 0 rz 168 deg; joints []
  MoveL (T451) to (-6.95, -39.39, 50) mm, rotated rx -90 ry 0 rz 170 deg; joints []
  MoveL (T452) to (-5.57, -39.61, 40) mm, rotated rx -90 ry 0 rz 172 deg; joints []
  MoveL (T453) to (-4.18, -39.78, 30) mm, rotated rx -90 ry 0 rz 174 deg; joints []
  MoveL (T454) to (-2.79, -39.9, 20) mm, rotated rx -90 ry 0 rz 176 deg; joints []
  MoveL (T455) to (-1.4, -39.98, 10) mm, rotated rx -90 ry 0 rz 178 deg; joints []
  MoveL (T456) to (0, -40, 0) mm, rotated rx -90 ry 0 rz 180 deg; joints []
  MoveL (T457) to (0, -100, 0) mm, rotated rx -90 ry 0 rz 180 deg; joints []
  MoveL (T458) to (17.36, -98.48, 0) mm, rotated rx -90 ry 0 rz -170 deg; joints []
  MoveL (T459) to (34.2, -93.97, 0) mm, rotated rx -90 ry 0 rz -160 deg; joints []
  MoveL (T460) to (50, -86.6, 0) mm, rotated rx -90 ry 0 rz -150 deg; joints []
  MoveL (T461) to (64.28, -76.6, 0) mm, rotated rx -90 ry 0 rz -140 deg; joints []
  MoveL (T462) to (76.6, -64.28, 0) mm, rotated rx -90 ry 0 rz -130 deg; joints []
  MoveL (T463) to (86.6, -50, 0) mm, rotated rx -90 ry 0 rz -120 deg; joints []
  MoveL (T464) to (34.64, -20, 0) mm, rotated rx -90 ry 0 rz -120 deg; joints []
  MoveL (T465) to (30.64, -25.71, 1.67) mm, rotated rx -90 ry 0 rz -130 deg; joints []
  MoveL (T466) to (25.71, -30.64, 3.33) mm, rotated rx -90 ry 0 rz -140 deg; joints []
  MoveL (T467) to (20, -34.64, 5) mm, rotated rx -90 ry 0 rz -150 deg; joints []
  MoveL (T468) to (13.68, -37.59, 6.67) mm, rotated rx -90 ry 0 rz -160 deg; joints []
  MoveL (T469) to (6.95, -39.39, 8.33) mm, rotated rx -90 ry 0 rz -170 deg; joints []
  MoveL (T470) to (0, -40, 10) mm, rotated rx -90 ry 0 rz 180 deg; joints []
  MoveL (T471) to (0, -100, 10) mm, rotated rx -90 ry 0 rz 180 deg; joints []
  MoveL (T472) to (17.36, -98.48, 10) mm, rotated rx -90 ry 0 rz -170 deg; joints []
  MoveL (T473) to (34.2, -93.97, 10) mm, rotated rx -90 ry 0 rz -160 deg; joints []
  MoveL (T474) to (50, -86.6, 10) mm, rotated rx -90 ry 0 rz -150 deg; joints []
  MoveL (T475) to (64.28, -76.6, 10) mm, rotated rx -90 ry 0 rz -140 deg; joints []
  MoveL (T476) to (76.6, -64.28, 10) mm, rotated rx -90 ry 0 rz -130 deg; joints []
  MoveL (T477) to (86.6, -50, 10) mm, rotated rx -90 ry 0 rz -120 deg; joints []
  MoveL (T478) to (34.64, -20, 10) mm, rotated rx -90 ry 0 rz -120 deg; joints []
  MoveL (T479) to (30.64, -25.71, 11.67) mm, rotated rx -90 ry 0 rz -130 deg; joints []
  MoveL (T480) to (25.71, -30.64, 13.33) mm, rotated rx -90 ry 0 rz -140 deg; joints []
  MoveL (T481) to (20, -34.64, 15) mm, rotated rx -90 ry 0 rz -150 deg; joints []
  MoveL (T482) to (13.68, -37.59, 16.67) mm, rotated rx -90 ry 0 rz -160 deg; joints []
  MoveL (T483) to (6.95, -39.39, 18.33) mm, rotated rx -90 ry 0 rz -170 deg; joints []
  MoveL (T484) to (0, -40, 20) mm, rotated rx -90 ry 0 rz 180 deg; joints []
  MoveL (T485) to (0, -100, 20) mm, rotated rx -90 ry 0 rz 180 deg; joints []
  MoveL (T486) to (17.36, -98.48, 20) mm, rotated rx -90 ry 0 rz -170 deg; joints []
  MoveL (T487) to (34.2, -93.97, 20) mm, rotated rx -90 ry 0 rz -160 deg; joints []
  MoveL (T488) to (50, -86.6, 20) mm, rotated rx -90 ry 0 rz -150 deg; joints []
  MoveL (T489) to (64.28, -76.6, 20) mm, rotated rx -90 ry 0 rz -140 deg; joints []
  MoveL (T490) to (76.6, -64.28, 20) mm, rotated rx -90 ry 0 rz -130 deg; joints []
  MoveL (T491) to (86.6, -50, 20) mm, rotated rx -90 ry 0 rz -120 deg; joints []
  MoveL (T492) to (34.64, -20, 20) mm, rotated rx -90 ry 0 rz -120 deg; joints []
  MoveL (T493) to (30.64, -25.71, 21.67) mm, rotated rx -90 ry 0 rz -130 deg; joints []
  MoveL (T494) to (25.71, -30.64, 23.33) mm, rotated rx -90 ry 0 rz -140 deg; joints []
  MoveL (T495) to (20, -34.64, 25) mm, rotated rx -90 ry 0 rz -150 deg; joints []
  MoveL (T496) to (13.68, -37.59, 26.67) mm, rotated rx -90 ry 0 rz -160 deg; joints []
  MoveL (T497) to (6.95, -39.39, 28.33) mm, rotated rx -90 ry 0 rz -170 deg; joints []
  MoveL (T498) to (0, -40, 30) mm, rotated rx -90 ry 0 rz 180 deg; joints []
  MoveL (T499) to (0, -100, 30) mm, rotated rx -90 ry 0 rz 180 deg; joints []
  MoveL (T500) to (17.36, -98.48, 30) mm, rotated rx -90 ry 0 rz -170 deg; joints []
  MoveL (T501) to (34.2, -93.97, 30) mm, rotated rx -90 ry 0 rz -160 deg; joints []
  MoveL (T502) to (50, -86.6, 30) mm, rotated rx -90 ry 0 rz -150 deg; joints []
  MoveL (T503) to (64.28, -76.6, 30) mm, rotated rx -90 ry 0 rz -140 deg; joints []
  MoveL (T504) to (76.6, -64.28, 30) mm, rotated rx -90 ry 0 rz -130 deg; joints []
  MoveL (T505) to (86.6, -50, 30) mm, rotated rx -90 ry 0 rz -120 deg; joints []
  MoveL (T506) to (34.64, -20, 30) mm, rotated rx -90 ry 0 rz -120 deg; joints []
  MoveL (T507) to (30.64, -25.71, 31.67) mm, rotated rx -90 ry 0 rz -130 deg; joints []
  MoveL (T508) to (25.71, -30.64, 33.33) mm, rotated rx -90 ry 0 rz -140 deg; joints []
  MoveL (T509) to (20, -34.64, 35) mm, rotated rx -90 ry 0 rz -150 deg; joints []
  MoveL (T510) to (13.68, -37.59, 36.67) mm, rotated rx -90 ry 0 rz -160 deg; joints []
  MoveL (T511) to (6.95, -39.39, 38.33) mm, rotated rx -90 ry 0 rz -170 deg; joints []
  MoveL (T512) to (0, -40, 40) mm, rotated rx -90 ry 0 rz 180 deg; joints []
  MoveL (T513) to (0, -100, 40) mm, rotated rx -90 ry 0 rz 180 deg; joints []
  MoveL (T514) to (17.36, -98.48, 40) mm, rotated rx -90 ry 0 rz -170 deg; joints []
  MoveL (T515) to (34.2, -93.97, 40) mm, rotated rx -90 ry 0 rz -160 deg; joints []
  MoveL (T516) to (50, -86.6, 40) mm, rotated rx -90 ry 0 rz -150 deg; joints []
  MoveL (T517) to (64.28, -76.6, 40) mm, rotated rx -90 ry 0 rz -140 deg; joints []
  MoveL (T518) to (76.6, -64.28, 40) mm, rotated rx -90 ry 0 rz -130 deg; joints []
  MoveL (T519) to (86.6, -50, 40) mm, rotated rx -90 ry 0 rz -120 deg; joints []
  MoveL (T520) to (34.64, -20, 40) mm, rotated rx -90 ry 0 rz -120 deg; joints []
  MoveL (T521) to (30.64, -25.71, 41.67) mm, rotated rx -90 ry 0 rz -130 deg; joints []
  MoveL (T522) to (25.71, -30.64, 43.33) mm, rotated rx -90 ry 0 rz -140 deg; joints []
  MoveL (T523) to (20, -34.64, 45) mm, rotated rx -90 ry 0 rz -150 deg; joints []
  MoveL (T524) to (13.68, -37.59, 46.67) mm, rotated rx -90 ry 0 rz -160 deg; joints []
  MoveL (T525) to (6.95, -39.39, 48.33) mm, rotated rx -90 ry 0 rz -170 deg; joints []
  MoveL (T526) to (0, -40, 50) mm, rotated rx -90 ry 0 rz 180 deg; joints []
  MoveL (T527) to (0, -100, 50) mm, rotated rx -90 ry 0 rz 180 deg; joints []
  MoveL (T528) to (17.36, -98.48, 50) mm, rotated rx -90 ry 0 rz -170 deg; joints []
  MoveL (T529) to (34.2, -93.97, 50) mm, rotated rx -90 ry 0 rz -160 deg; joints []
  MoveL (T530) to (50, -86.6, 50) mm, rotated rx -90 ry 0 rz -150 deg; joints []
  MoveL (T531) to (64.28, -76.6, 50) mm, rotated rx -90 ry 0 rz -140 deg; joints []
  MoveL (T532) to (76.6, -64.28, 50) mm, rotated rx -90 ry 0 rz -130 deg; joints []
  MoveL (T533) to (86.6, -50, 50) mm, rotated rx -90 ry 0 rz -120 deg; joints []
  MoveL (T534) to (34.64, -20, 50) mm, rotated rx -90 ry 0 rz -120 deg; joints []
  MoveL (T535) to (30.64, -25.71, 51.67) mm, rotated rx -90 ry 0 rz -130 deg; joints []
  MoveL (T536) to (25.71, -30.64, 53.33) mm, rotated rx -90 ry 0 rz -140 deg; joints []
  MoveL (T537) to (20, -34.64, 55) mm, rotated rx -90 ry 0 rz -150 deg; joints []
  MoveL (T538) to (13.68, -37.59, 56.67) mm, rotated rx -90 ry 0 rz -160 deg; joints []
  MoveL (T539) to (6.95, -39.39, 58.33) mm, rotated rx -90 ry 0 rz -170 deg; joints []
  MoveL (T540) to (0, -40, 60) mm, rotated rx -90 ry 0 rz 180 deg; joints []
  MoveL (T541) to (0, -100, 60) mm, rotated rx -90 ry 0 rz 180 deg; joints []
  MoveL (T542) to (17.36, -98.48, 60) mm, rotated rx -90 ry 0 rz -170 deg; joints []
  MoveL (T543) to (34.2, -93.97, 60) mm, rotated rx -90 ry 0 rz -160 deg; joints []
  MoveL (T544) to (50, -86.6, 60) mm, rotated rx -90 ry 0 rz -150 deg; joints []
  MoveL (T545) to (64.28, -76.6, 60) mm, rotated rx -90 ry 0 rz -140 deg; joints []
  MoveL (T546) to (76.6, -64.28, 60) mm, rotated rx -90 ry 0 rz -130 deg; joints []
  MoveL (T547) to (86.6, -50, 60) mm, rotated rx -90 ry 0 rz -120 deg; joints []
  MoveL (T548) to (34.64, -20, 60) mm, rotated rx -90 ry 0 rz -120 deg; joints []
  MoveL (T549) to (30.64, -25.71, 61.67) mm, rotated rx -90 ry 0 rz -130 deg; joints []
  MoveL (T550) to (25.71, -30.64, 63.33) mm, rotated rx -90 ry 0 rz -140 deg; joints []
  MoveL (T551) to (20, -34.64, 65) mm, rotated rx -90 ry 0 rz -150 deg; joints []
  MoveL (T552) to (13.68, -37.59, 66.67) mm, rotated rx -90 ry 0 rz -160 deg; joints []
  MoveL (T553) to (6.95, -39.39, 68.33) mm, rotated rx -90 ry 0 rz -170 deg; joints []
  MoveL (T554) to (0, -40, 70) mm, rotated rx -90 ry 0 rz 180 deg; joints []
  MoveL (T555) to (0, -100, 70) mm, rotated rx -90 ry 0 rz 180 deg; joints []
  MoveL (T556) to (17.36, -98.48, 70) mm, rotated rx -90 ry 0 rz -170 deg; joints []
  MoveL (T557) to (34.2, -93.97, 70) mm, rotated rx -90 ry 0 rz -160 deg; joints []
  MoveL (T558) to (50, -86.6, 70) mm, rotated rx -90 ry 0 rz -150 deg; joints []
  MoveL (T559) to (64.28, -76.6, 70) mm, rotated rx -90 ry 0 rz -140 deg; joints []
  MoveL (T560) to (76.6, -64.28, 70) mm, rotated rx -90 ry 0 rz -130 deg; joints []
  MoveL (T561) to (86.6, -50, 70) mm, rotated rx -90 ry 0 rz -120 deg; joints []
  MoveL (T562) to (34.64, -20, 70) mm, rotated rx -90 ry 0 rz -120 deg; joints []
  MoveL (T563) to (30.64, -25.71, 71.67) mm, rotated rx -90 ry 0 rz -130 deg; joints []
  MoveL (T564) to (25.71, -30.64, 73.33) mm, rotated rx -90 ry 0 rz -140 deg; joints []
  MoveL (T565) to (20, -34.64, 75) mm, rotated rx -90 ry 0 rz -150 deg; joints []
  MoveL (T566) to (13.68, -37.59, 76.67) mm, rotated rx -90 ry 0 rz -160 deg; joints []
  MoveL (T567) to (6.95, -39.39, 78.33) mm, rotated rx -90 ry 0 rz -170 deg; joints []
  MoveL (T568) to (0, -40, 80) mm, rotated rx -90 ry 0 rz 180 deg; joints []
  MoveL (T569) to (0, -100, 80) mm, rotated rx -90 ry 0 rz 180 deg; joints []
  MoveL (T570) to (17.36, -98.48, 80) mm, rotated rx -90 ry 0 rz -170 deg; joints []
  MoveL (T571) to (34.2, -93.97, 80) mm, rotated rx -90 ry 0 rz -160 deg; joints []
  MoveL (T572) to (50, -86.6, 80) mm, rotated rx -90 ry 0 rz -150 deg; joints []
  MoveL (T573) to (64.28, -76.6, 80) mm, rotated rx -90 ry 0 rz -140 deg; joints []
  MoveL (T574) to (76.6, -64.28, 80) mm, rotated rx -90 ry 0 rz -130 deg; joints []
  MoveL (T575) to (86.6, -50, 80) mm, rotated rx -90 ry 0 rz -120 deg; joints []
  MoveL (T576) to (34.64, -20, 80) mm, rotated rx -90 ry 0 rz -120 deg; joints []
  MoveL (T577) to (30.64, -25.71, 81.67) mm, rotated rx -90 ry 0 rz -130 deg; joints []
  MoveL (T578) to (25.71, -30.64, 83.33) mm, rotated rx -90 ry 0 rz -140 deg; joints []
  MoveL (T579) to (20, -34.64, 85) mm, rotated rx -90 ry 0 rz -150 deg; joints []
  MoveL (T580) to (13.68, -37.59, 86.67) mm, rotated rx -90 ry 0 rz -160 deg; joints []
  MoveL (T581) to (6.95, -39.39, 88.33) mm, rotated rx -90 ry 0 rz -170 deg; joints []
  MoveL (T582) to (0, -40, 90) mm, rotated rx -90 ry 0 rz 180 deg; joints []
  MoveL (T583) to (0, -100, 90) mm, rotated rx -90 ry 0 rz 180 deg; joints []
  MoveL (T584) to (17.36, -98.48, 90) mm, rotated rx -90 ry 0 rz -170 deg; joints []
  MoveL (T585) to (34.2, -93.97, 90) mm, rotated rx -90 ry 0 rz -160 deg; joints []
  MoveL (T586) to (50, -86.6, 90) mm, rotated rx -90 ry 0 rz -150 deg; joints []
  MoveL (T587) to (64.28, -76.6, 90) mm, rotated rx -90 ry 0 rz -140 deg; joints []
  MoveL (T588) to (76.6, -64.28, 90) mm, rotated rx -90 ry 0 rz -130 deg; joints []
  MoveL (T589) to (86.6, -50, 90) mm, rotated rx -90 ry 0 rz -120 deg; joints []
  MoveL (T590) to (34.64, -20, 90) mm, rotated rx -90 ry 0 rz -120 deg; joints []
  MoveL (T591) to (30.64, -25.71, 91.67) mm, rotated rx -90 ry 0 rz -130 deg; joints []
  MoveL (T592) to (25.71, -30.64, 93.33) mm, rotated rx -90 ry 0 rz -140 deg; joints []
  MoveL (T593) to (20, -34.64, 95) mm, rotated rx -90 ry 0 rz -150 deg; joints []
  MoveL (T594) to (13.68, -37.59, 96.67) mm, rotated rx -90 ry 0 rz -160 deg; joints []
  MoveL (T595) to (6.95, -39.39, 98.33) mm, rotated rx -90 ry 0 rz -170 deg; joints []
  MoveL (T596) to (0, -40, 100) mm, rotated rx -90 ry 0 rz 180 deg; joints []
  MoveL (T597) to (0, -100, 100) mm, rotated rx -90 ry 0 rz 180 deg; joints []
  MoveL (T598) to (17.36, -98.48, 100) mm, rotated rx -90 ry 0 rz -170 deg; joints []
  MoveL (T599) to (34.2, -93.97, 100) mm, rotated rx -90 ry 0 rz -160 deg; joints []
  MoveL (T600) to (50, -86.6, 100) mm, rotated rx -90 ry 0 rz -150 deg; joints []
  MoveL (T601) to (64.28, -76.6, 100) mm, rotated rx -90 ry 0 rz -140 deg; joints []
  MoveL (T602) to (76.6, -64.28, 100) mm, rotated rx -90 ry 0 rz -130 deg; joints []
  MoveL (T603) to (86.6, -50, 100) mm, rotated rx -90 ry 0 rz -120 deg; joints []
  MoveL (T604) to (34.64, -20, 100) mm, rotated rx -90 ry 0 rz -120 deg; joints []
  MoveL (T605) to (30.64, -25.71, 101.67) mm, rotated rx -90 ry 0 rz -130 deg; joints []
  MoveL (T606) to (25.71, -30.64, 103.33) mm, rotated rx -90 ry 0 rz -140 deg; joints []
  MoveL (T607) to (20, -34.64, 105) mm, rotated rx -90 ry 0 rz -150 deg; joints []
  MoveL (T608) to (13.68, -37.59, 106.67) mm, rotated rx -90 ry 0 rz -160 deg; joints []
  MoveL (T609) to (6.95, -39.39, 108.33) mm, rotated rx -90 ry 0 rz -170 deg; joints []
  MoveL (T610) to (0, -40, 110) mm, rotated rx -90 ry 0 rz 180 deg; joints []
  MoveL (T611) to (0, -100, 110) mm, rotated rx -90 ry 0 rz 180 deg; joints []
  MoveL (T612) to (17.36, -98.48, 110) mm, rotated rx -90 ry 0 rz -170 deg; joints []
  MoveL (T613) to (34.2, -93.97, 110) mm, rotated rx -90 ry 0 rz -160 deg; joints []
  MoveL (T614) to (50, -86.6, 110) mm, rotated rx -90 ry 0 rz -150 deg; joints []
  MoveL (T615) to (64.28, -76.6, 110) mm, rotated rx -90 ry 0 rz -140 deg; joints []
  MoveL (T616) to (76.6, -64.28, 110) mm, rotated rx -90 ry 0 rz -130 deg; joints []
  MoveL (T617) to (86.6, -50, 110) mm, rotated rx -90 ry 0 rz -120 deg; joints []
  MoveL (T618) to (34.64, -20, 110) mm, rotated rx -90 ry 0 rz -120 deg; joints []
  MoveL (T619) to (30.64, -25.71, 111.67) mm, rotated rx -90 ry 0 rz -130 deg; joints []
  MoveL (T620) to (25.71, -30.64, 113.33) mm, rotated rx -90 ry 0 rz -140 deg; joints []
  MoveL (T621) to (20, -34.64, 115) mm, rotated rx -90 ry 0 rz -150 deg; joints []
  MoveL (T622) to (13.68, -37.59, 116.67) mm, rotated rx -90 ry 0 rz -160 deg; joints []
  MoveL (T623) to (6.95, -39.39, 118.33) mm, rotated rx -90 ry 0 rz -170 deg; joints []
  MoveL (T624) to (0, -40, 120) mm, rotated rx -90 ry 0 rz 180 deg; joints []
  MoveL (T625) to (0, -100, 120) mm, rotated rx -90 ry 0 rz 180 deg; joints []
  MoveL (T626) to (17.36, -98.48, 120) mm, rotated rx -90 ry 0 rz -170 deg; joints []
  MoveL (T627) to (34.2, -93.97, 120) mm, rotated rx -90 ry 0 rz -160 deg; joints []
  MoveL (T628) to (50, -86.6, 120) mm, rotated rx -90 ry 0 rz -150 deg; joints []
  MoveL (T629) to (64.28, -76.6, 120) mm, rotated rx -90 ry 0 rz -140 deg; joints []
  MoveL (T630) to (76.6, -64.28, 120) mm, rotated rx -90 ry 0 rz -130 deg; joints []
  MoveL (T631) to (86.6, -50, 120) mm, rotated rx -90 ry 0 rz -120 deg; joints []
  MoveL (T632) to (34.64, -20, 120) mm, rotated rx -90 ry 0 rz -120 deg; joints []
  MoveL (T633) to (30.64, -25.71, 121.67) mm, rotated rx -90 ry 0 rz -130 deg; joints []
  MoveL (T634) to (25.71, -30.64, 123.33) mm, rotated rx -90 ry 0 rz -140 deg; joints []
  MoveL (T635) to (20, -34.64, 125) mm, rotated rx -90 ry 0 rz -150 deg; joints []
  MoveL (T636) to (13.68, -37.59, 126.67) mm, rotated rx -90 ry 0 rz -160 deg; joints []
  MoveL (T637) to (6.95, -39.39, 128.33) mm, rotated rx -90 ry 0 rz -170 deg; joints []
  MoveL (T638) to (0, -40, 130) mm, rotated rx -90 ry 0 rz 180 deg; joints []
  MoveL (T639) to (0, -100, 130) mm, rotated rx -90 ry 0 rz 180 deg; joints []
  MoveL (T640) to (17.36, -98.48, 130) mm, rotated rx -90 ry 0 rz -170 deg; joints []
  MoveL (T641) to (34.2, -93.97, 130) mm, rotated rx -90 ry 0 rz -160 deg; joints []
  MoveL (T642) to (50, -86.6, 130) mm, rotated rx -90 ry 0 rz -150 deg; joints []
  MoveL (T643) to (64.28, -76.6, 130) mm, rotated rx -90 ry 0 rz -140 deg; joints []
  MoveL (T644) to (76.6, -64.28, 130) mm, rotated rx -90 ry 0 rz -130 deg; joints []
  MoveL (T645) to (86.6, -50, 130) mm, rotated rx -90 ry 0 rz -120 deg; joints []
  MoveL (T646) to (34.64, -20, 130) mm, rotated rx -90 ry 0 rz -120 deg; joints []
  MoveL (T647) to (30.64, -25.71, 131.67) mm, rotated rx -90 ry 0 rz -130 deg; joints []
  MoveL (T648) to (25.71, -30.64, 133.33) mm, rotated rx -90 ry 0 rz -140 deg; joints []
  MoveL (T649) to (20, -34.64, 135) mm, rotated rx -90 ry 0 rz -150 deg; joints []
  MoveL (T650) to (13.68, -37.59, 136.67) mm, rotated rx -90 ry 0 rz -160 deg; joints []
  MoveL (T651) to (6.95, -39.39, 138.33) mm, rotated rx -90 ry 0 rz -170 deg; joints []
  MoveL (T652) to (0, -40, 140) mm, rotated rx -90 ry 0 rz 180 deg; joints []
  MoveL (T653) to (0, -100, 140) mm, rotated rx -90 ry 0 rz 180 deg; joints []
  MoveL (T654) to (17.36, -98.48, 140) mm, rotated rx -90 ry 0 rz -170 deg; joints []
  MoveL (T655) to (34.2, -93.97, 140) mm, rotated rx -90 ry 0 rz -160 deg; joints []
  MoveL (T656) to (50, -86.6, 140) mm, rotated rx -90 ry 0 rz -150 deg; joints []
  MoveL (T657) to (64.28, -76.6, 140) mm, rotated rx -90 ry 0 rz -140 deg; joints []
  MoveL (T658) to (76.6, -64.28, 140) mm, rotated rx -90 ry 0 rz -130 deg; joints []
  MoveL (T659) to (86.6, -50, 140) mm, rotated rx -90 ry 0 rz -120 deg; joints []
  MoveL (T660) to (34.64, -20, 140) mm, rotated rx -90 ry 0 rz -120 deg; joints []
  MoveL (T661) to (30.64, -25.71, 141.67) mm, rotated rx -90 ry 0 rz -130 deg; joints []
  MoveL (T662) to (25.71, -30.64, 143.33) mm, rotated rx -90 ry 0 rz -140 deg; joints []
  MoveL (T663) to (20, -34.64, 145) mm, rotated rx -90 ry 0 rz -150 deg; joints []
  MoveL (T664) to (13.68, -37.59, 146.67) mm, rotated rx -90 ry 0 rz -160 deg; joints []
  MoveL (T665) to (6.95, -39.39, 148.33) mm, rotated rx -90 ry 0 rz -170 deg; joints []
  MoveL (T666) to (0, -40, 150) mm, rotated rx -90 ry 0 rz 180 deg; joints []
  MoveL (T667) to (0, -100, 150) mm, rotated rx -90 ry 0 rz 180 deg; joints []
  MoveL (T668) to (17.36, -98.48, 150) mm, rotated rx -90 ry 0 rz -170 deg; joints []
  MoveL (T669) to (34.2, -93.97, 150) mm, rotated rx -90 ry 0 rz -160 deg; joints []
  MoveL (T670) to (50, -86.6, 150) mm, rotated rx -90 ry 0 rz -150 deg; joints []
  MoveL (T671) to (64.28, -76.6, 150) mm, rotated rx -90 ry 0 rz -140 deg; joints []
  MoveL (T672) to (76.6, -64.28, 150) mm, rotated rx -90 ry 0 rz -130 deg; joints []
  MoveL (T673) to (86.6, -50, 150) mm, rotated rx -90 ry 0 rz -120 deg; joints []
  MoveL (T674) to (34.64, -20, 150) mm, rotated rx -90 ry 0 rz -120 deg; joints []
  MoveL (T675) to (34.64, -20, 140) mm, rotated rx -90 ry 0 rz -120 deg; joints []
  MoveL (T676) to (34.64, -20, 130) mm, rotated rx -90 ry 0 rz -120 deg; joints []
  MoveL (T677) to (34.64, -20, 120) mm, rotated rx -90 ry 0 rz -120 deg; joints []
  MoveL (T678) to (34.64, -20, 110) mm, rotated rx -90 ry 0 rz -120 deg; joints []
  MoveL (T679) to (34.64, -20, 100) mm, rotated rx -90 ry 0 rz -120 deg; joints []
  MoveL (T680) to (34.64, -20, 90) mm, rotated rx -90 ry 0 rz -120 deg; joints []
  MoveL (T681) to (34.64, -20, 80) mm, rotated rx -90 ry 0 rz -120 deg; joints []
  MoveL (T682) to (34.64, -20, 70) mm, rotated rx -90 ry 0 rz -120 deg; joints []
  MoveL (T683) to (34.64, -20, 60) mm, rotated rx -90 ry 0 rz -120 deg; joints []
  MoveL (T684) to (34.64, -20, 50) mm, rotated rx -90 ry 0 rz -120 deg; joints []
  MoveL (T685) to (34.64, -20, 40) mm, rotated rx -90 ry 0 rz -120 deg; joints []
  MoveL (T686) to (34.64, -20, 30) mm, rotated rx -90 ry 0 rz -120 deg; joints []
  MoveL (T687) to (34.64, -20, 20) mm, rotated rx -90 ry 0 rz -120 deg; joints []
  MoveL (T688) to (34.64, -20, 10) mm, rotated rx -90 ry 0 rz -120 deg; joints []
  MoveL (T689) to (34.64, -20, 0) mm, rotated rx -90 ry 0 rz -120 deg; joints []
  MoveL (T690) to (86.6, -50, 0) mm, rotated rx -90 ry 0 rz -120 deg; joints []
  MoveL (T691) to (86.6, -50, 10) mm, rotated rx -90 ry 0 rz -120 deg; joints []
  MoveL (T692) to (86.6, -50, 20) mm, rotated rx -90 ry 0 rz -120 deg; joints []
  MoveL (T693) to (86.6, -50, 30) mm, rotated rx -90 ry 0 rz -120 deg; joints []
  MoveL (T694) to (86.6, -50, 40) mm, rotated rx -90 ry 0 rz -120 deg; joints []
  MoveL (T695) to (86.6, -50, 50) mm, rotated rx -90 ry 0 rz -120 deg; joints []
  MoveL (T696) to (86.6, -50, 60) mm, rotated rx -90 ry 0 rz -120 deg; joints []
  MoveL (T697) to (86.6, -50, 70) mm, rotated rx -90 ry 0 rz -120 deg; joints []
  MoveL (T698) to (86.6, -50, 80) mm, rotated rx -90 ry 0 rz -120 deg; joints []
  MoveL (T699) to (86.6, -50, 90) mm, rotated rx -90 ry 0 rz -120 deg; joints []
  MoveL (T700) to (86.6, -50, 100) mm, rotated rx -90 ry 0 rz -120 deg; joints []
  MoveL (T701) to (86.6, -50, 110) mm, rotated rx -90 ry 0 rz -120 deg; joints []
  MoveL (T702) to (86.6, -50, 120) mm, rotated rx -90 ry 0 rz -120 deg; joints []
  MoveL (T703) to (86.6, -50, 130) mm, rotated rx -90 ry 0 rz -120 deg; joints []
  MoveL (T704) to (86.6, -50, 140) mm, rotated rx -90 ry 0 rz -120 deg; joints []
  MoveL (T705) to (86.6, -50, 150) mm, rotated rx -90 ry 0 rz -120 deg; joints []
  MoveL (T706) to (76.6, -64.28, 150) mm, rotated rx -90 ry 0 rz -130 deg; joints []
  MoveL (T707) to (64.28, -76.6, 150) mm, rotated rx -90 ry 0 rz -140 deg; joints []
  MoveL (T708) to (50, -86.6, 150) mm, rotated rx -90 ry 0 rz -150 deg; joints []
  MoveL (T709) to (34.2, -93.97, 150) mm, rotated rx -90 ry 0 rz -160 deg; joints []
  MoveL (T710) to (17.36, -98.48, 150) mm, rotated rx -90 ry 0 rz -170 deg; joints []
  MoveL (T711) to (0, -100, 150) mm, rotated rx -90 ry 0 rz 180 deg; joints []
  MoveL (T712) to (0, -100, 140) mm, rotated rx -90 ry 0 rz 180 deg; joints []
  MoveL (T713) to (0, -100, 130) mm, rotated rx -90 ry 0 rz 180 deg; joints []
  MoveL (T714) to (0, -100, 120) mm, rotated rx -90 ry 0 rz 180 deg; joints []
  MoveL (T715) to (0, -100, 110) mm, rotated rx -90 ry 0 rz 180 deg; joints []
  MoveL (T716) to (0, -100, 100) mm, rotated rx -90 ry 0 rz 180 deg; joints []
  MoveL (T717) to (0, -100, 90) mm, rotated rx -90 ry 0 rz 180 deg; joints []
  MoveL (T718) to (0, -100, 80) mm, rotated rx -90 ry 0 rz 180 deg; joints []
  MoveL (T719) to (0, -100, 70) mm, rotated rx -90 ry 0 rz 180 deg; joints []
  MoveL (T720) to (0, -100, 60) mm, rotated rx -90 ry 0 rz 180 deg; joints []
  MoveL (T721) to (0, -100, 50) mm, rotated rx -90 ry 0 rz 180 deg; joints []
  MoveL (T722) to (0, -100, 40) mm, rotated rx -90 ry 0 rz 180 deg; joints []
  MoveL (T723) to (0, -100, 30) mm, rotated rx -90 ry 0 rz 180 deg; joints []
  MoveL (T724) to (0, -100, 20) mm, rotated rx -90 ry 0 rz 180 deg; joints []
  MoveL (T725) to (0, -100, 10) mm, rotated rx -90 ry 0 rz 180 deg; joints []
  MoveL (T726) to (0, -100, 0) mm, rotated rx -90 ry 0 rz 180 deg; joints []
  MoveL (T727) to (17.36, -98.48, 0) mm, rotated rx -90 ry 0 rz -170 deg; joints []
  MoveL (T728) to (34.2, -93.97, 0) mm, rotated rx -90 ry 0 rz -160 deg; joints []
  MoveL (T729) to (50, -86.6, 0) mm, rotated rx -90 ry 0 rz -150 deg; joints []
  MoveL (T730) to (64.28, -76.6, 0) mm, rotated rx -90 ry 0 rz -140 deg; joints []
  MoveL (T731) to (76.6, -64.28, 0) mm, rotated rx -90 ry 0 rz -130 deg; joints []
  MoveL (T732) to (86.6, -50, 0) mm, rotated rx -90 ry 0 rz -120 deg; joints []
  MoveL (T733) to (34.64, -20, 0) mm, rotated rx -90 ry 0 rz -120 deg; joints []
  MoveL (T734) to (30.64, -25.71, 0) mm, rotated rx -90 ry 0 rz -130 deg; joints []
  MoveL (T735) to (25.71, -30.64, 0) mm, rotated rx -90 ry 0 rz -140 deg; joints []
  MoveL (T736) to (20, -34.64, 0) mm, rotated rx -90 ry 0 rz -150 deg; joints []
  MoveL (T737) to (13.68, -37.59, 0) mm, rotated rx -90 ry 0 rz -160 deg; joints []
  MoveL (T738) to (6.95, -39.39, 0) mm, rotated rx -90 ry 0 rz -170 deg; joints []
  MoveL (T739) to (0, -40, 0) mm, rotated rx -90 ry 0 rz 180 deg; joints []
  MoveL (T740) to (-6.95, -39.39, 0) mm, rotated rx -90 ry 0 rz 170 deg; joints []
  MoveL (T741) to (-13.68, -37.59, 0) mm, rotated rx -90 ry 0 rz 160 deg; joints []
  MoveL (T742) to (-20, -34.64, 0) mm, rotated rx -90 ry 0 rz 150 deg; joints []
  MoveL (T743) to (-50, -86.6, 0) mm, rotated rx -90 ry 0 rz 150 deg; joints []
  MoveL (T744) to (-50, -86.6, 10) mm, rotated rx -90 ry 0 rz 150 deg; joints []
  MoveL (T745) to (-50, -86.6, 20) mm, rotated rx -90 ry 0 rz 150 deg; joints []
  MoveL (T746) to (-50, -86.6, 30) mm, rotated rx -90 ry 0 rz 150 deg; joints []
  MoveL (T747) to (-50, -86.6, 40) mm, rotated rx -90 ry 0 rz 150 deg; joints []
  MoveL (T748) to (-50, -86.6, 50) mm, rotated rx -90 ry 0 rz 150 deg; joints []
  MoveL (T749) to (-50, -86.6, 60) mm, rotated rx -90 ry 0 rz 150 deg; joints []
  MoveL (T750) to (-50, -86.6, 70) mm, rotated rx -90 ry 0 rz 150 deg; joints []
  MoveL (T751) to (-50, -86.6, 80) mm, rotated rx -90 ry 0 rz 150 deg; joints []
  MoveL (T752) to (-50, -86.6, 90) mm, rotated rx -90 ry 0 rz 150 deg; joints []
  MoveL (T753) to (-50, -86.6, 100) mm, rotated rx -90 ry 0 rz 150 deg; joints []
  MoveL (T754) to (-50, -86.6, 110) mm, rotated rx -90 ry 0 rz 150 deg; joints []
  MoveL (T755) to (-50, -86.6, 120) mm, rotated rx -90 ry 0 rz 150 deg; joints []
  MoveL (T756) to (-50, -86.6, 130) mm, rotated rx -90 ry 0 rz 150 deg; joints []
  MoveL (T757) to (-50, -86.6, 140) mm, rotated rx -90 ry 0 rz 150 deg; joints []
  MoveL (T758) to (-50, -86.6, 150) mm, rotated rx -90 ry 0 rz 150 deg; joints []
  MoveL (T759) to (-64.28, -76.6, 150) mm, rotated rx -90 ry 0 rz 140 deg; joints []
  MoveL (T760) to (-76.6, -64.28, 150) mm, rotated rx -90 ry 0 rz 130 deg; joints []
  MoveL (T761) to (-86.6, -50, 150) mm, rotated rx -90 ry 0 rz 120 deg; joints []
  MoveL (T762) to (-93.97, -34.2, 150) mm, rotated rx -90 ry 0 rz 110 deg; joints []
  MoveL (T763) to (-98.48, -17.36, 150) mm, rotated rx -90 ry 0 rz 100 deg; joints []
  MoveL (T764) to (-100, 0, 150) mm, rotated rx -90 ry 0 rz 90 deg; joints []
  MoveL (T765) to (-100, 0, 140) mm, rotated rx -90 ry 0 rz 90 deg; joints []
  MoveL (T766) to (-100, 0, 130) mm, rotated rx -90 ry 0 rz 90 deg; joints []
  MoveL (T767) to (-100, 0, 120) mm, rotated rx -90 ry 0 rz 90 deg; joints []
  MoveL (T768) to (-100, 0, 110) mm, rotated rx -90 ry 0 rz 90 deg; joints []
  MoveL (T769) to (-100, 0, 100) mm, rotated rx -90 ry 0 rz 90 deg; joints []
  MoveL (T770) to (-100, 0, 90) mm, rotated rx -90 ry 0 rz 90 deg; joints []
  MoveL (T771) to (-100, 0, 80) mm, rotated rx -90 ry 0 rz 90 deg; joints []
  MoveL (T772) to (-100, 0, 70) mm, rotated rx -90 ry 0 rz 90 deg; joints []
  MoveL (T773) to (-100, 0, 60) mm, rotated rx -90 ry 0 rz 90 deg; joints []
  MoveL (T774) to (-100, 0, 50) mm, rotated rx -90 ry 0 rz 90 deg; joints []
  MoveL (T775) to (-100, 0, 40) mm, rotated rx -90 ry 0 rz 90 deg; joints []
  MoveL (T776) to (-100, 0, 30) mm, rotated rx -90 ry 0 rz 90 deg; joints []
  MoveL (T777) to (-100, 0, 20) mm, rotated rx -90 ry 0 rz 90 deg; joints []
  MoveL (T778) to (-100, 0, 10) mm, rotated rx -90 ry 0 rz 90 deg; joints []
  MoveL (T779) to (-100, 0, 0) mm, rotated rx -90 ry 0 rz 90 deg; joints []
  MoveL (T780) to (-98.48, -17.36, 0) mm, rotated rx -90 ry 0 rz 100 deg; joints []
  MoveL (T781) to (-93.97, -34.2, 0) mm, rotated rx -90 ry 0 rz 110 deg; joints []
  MoveL (T782) to (-86.6, -50, 0) mm, rotated rx -90 ry 0 rz 120 deg; joints []
  MoveL (T783) to (-76.6, -64.28, 0) mm, rotated rx -90 ry 0 rz 130 deg; joints []
  MoveL (T784) to (-64.28, -76.6, 0) mm, rotated rx -90 ry 0 rz 140 deg; joints []
  MoveL (T785) to (-50, -86.6, 0) mm, rotated rx -90 ry 0 rz 150 deg; joints []
  MoveL (T786) to (-20, -34.64, 0) mm, rotated rx -90 ry 0 rz 150 deg; joints []
  MoveL (T787) to (-25.71, -30.64, 0) mm, rotated rx -90 ry 0 rz 140 deg; joints []
  MoveL (T788) to (-30.64, -25.71, 0) mm, rotated rx -90 ry 0 rz 130 deg; joints []
  MoveL (T789) to (-34.64, -20, 0) mm, rotated rx -90 ry 0 rz 120 deg; joints []
  MoveL (T790) to (-37.59, -13.68, 0) mm, rotated rx -90 ry 0 rz 110 deg; joints []
  MoveL (T791) to (-39.39, -6.95, 0) mm, rotated rx -90 ry 0 rz 100 deg; joints []
  MoveL (T792) to (-40, 0, 0) mm, rotated rx -90 ry 0 rz 90 deg; joints []
  MoveL (T793) to (-39.39, 6.95, 0) mm, rotated rx -90 ry 0 rz 80 deg; joints []
  MoveL (T794) to (-37.59, 13.68, 0) mm, rotated rx -90 ry 0 rz 70 deg; joints []
  MoveL (T795) to (-34.64, 20, 0) mm, rotated rx -90 ry 0 rz 60 deg; joints []
  MoveL (T796) to (-86.6, 50, 0) mm, rotated rx -90 ry 0 rz 60 deg; joints []
  MoveL (T797) to (-86.6, 50, 10) mm, rotated rx -90 ry 0 rz 60 deg; joints []
  MoveL (T798) to (-86.6, 50, 20) mm, rotated rx -90 ry 0 rz 60 deg; joints []
  MoveL (T799) to (-86.6, 50, 30) mm, rotated rx -90 ry 0 rz 60 deg; joints []
  MoveL (T800) to (-86.6, 50, 40) mm, rotated rx -90 ry 0 rz 60 deg; joints []
  MoveL (T801) to (-86.6, 50, 50) mm, rotated rx -90 ry 0 rz 60 deg; joints []
  MoveL (T802) to (-86.6, 50, 60) mm, rotated rx -90 ry 0 rz 60 deg; joints []
  MoveL (T803) to (-86.6, 50, 70) mm, rotated rx -90 ry 0 rz 60 deg; joints []
  MoveL (T804) to (-86.6, 50, 80) mm, rotated rx -90 ry 0 rz 60 deg; joints []
  MoveL (T805) to (-86.6, 50, 90) mm, rotated rx -90 ry 0 rz 60 deg; joints []
  MoveL (T806) to (-86.6, 50, 100) mm, rotated rx -90 ry 0 rz 60 deg; joints []
  MoveL (T807) to (-86.6, 50, 110) mm, rotated rx -90 ry 0 rz 60 deg; joints []
  MoveL (T808) to (-86.6, 50, 120) mm, rotated rx -90 ry 0 rz 60 deg; joints []
  MoveL (T809) to (-86.6, 50, 130) mm, rotated rx -90 ry 0 rz 60 deg; joints []
  MoveL (T810) to (-86.6, 50, 140) mm, rotated rx -90 ry 0 rz 60 deg; joints []
  MoveL (T811) to (-86.6, 50, 150) mm, rotated rx -90 ry 0 rz 60 deg; joints []
  MoveL (T812) to (-76.6, 64.28, 150) mm, rotated rx -90 ry 0 rz 50 deg; joints []
  MoveL (T813) to (-64.28, 76.6, 150) mm, rotated rx -90 ry 0 rz 40 deg; joints []
  MoveL (T814) to (-50, 86.6, 150) mm, rotated rx -90 ry 0 rz 30 deg; joints []
  MoveL (T815) to (-34.2, 93.97, 150) mm, rotated rx -90 ry 0 rz 20 deg; joints []
  MoveL (T816) to (-17.36, 98.48, 150) mm, rotated rx -90 ry 0 rz 10 deg; joints []
  MoveL (T817) to (0, 100, 150) mm, rotated rx -90 ry 0 rz 0 deg; joints []
  MoveL (T818) to (0, 100, 140) mm, rotated rx -90 ry 0 rz 0 deg; joints []
  MoveL (T819) to (0, 100, 130) mm, rotated rx -90 ry 0 rz 0 deg; joints []
  MoveL (T820) to (0, 100, 120) mm, rotated rx -90 ry 0 rz 0 deg; joints []
  MoveL (T821) to (0, 100, 110) mm, rotated rx -90 ry 0 rz 0 deg; joints []
  MoveL (T822) to (0, 100, 100) mm, rotated rx -90 ry 0 rz 0 deg; joints []
  MoveL (T823) to (0, 100, 90) mm, rotated rx -90 ry 0 rz 0 deg; joints []
  MoveL (T824) to (0, 100, 80) mm, rotated rx -90 ry 0 rz 0 deg; joints []
  MoveL (T825) to (0, 100, 70) mm, rotated rx -90 ry 0 rz 0 deg; joints []
  MoveL (T826) to (0, 100, 60) mm, rotated rx -90 ry 0 rz 0 deg; joints []
  MoveL (T827) to (0, 100, 50) mm, rotated rx -90 ry 0 rz 0 deg; joints []
  MoveL (T828) to (0, 100, 40) mm, rotated rx -90 ry 0 rz 0 deg; joints []
  MoveL (T829) to (0, 100, 30) mm, rotated rx -90 ry 0 rz 0 deg; joints []
  MoveL (T830) to (0, 100, 20) mm, rotated rx -90 ry 0 rz 0 deg; joints []
  MoveL (T831) to (0, 100, 10) mm, rotated rx -90 ry 0 rz 0 deg; joints []
  MoveL (T832) to (0, 100, 0) mm, rotated rx -90 ry 0 rz 0 deg; joints []
  MoveL (T833) to (-17.36, 98.48, 0) mm, rotated rx -90 ry 0 rz 10 deg; joints []
  MoveL (T834) to (-34.2, 93.97, 0) mm, rotated rx -90 ry 0 rz 20 deg; joints []
  MoveL (T835) to (-50, 86.6, 0) mm, rotated rx -90 ry 0 rz 30 deg; joints []
  MoveL (T836) to (-64.28, 76.6, 0) mm, rotated rx -90 ry 0 rz 40 deg; joints []
  MoveL (T837) to (-76.6, 64.28, 0) mm, rotated rx -90 ry 0 rz 50 deg; joints []
  MoveL (T838) to (-86.6, 50, 0) mm, rotated rx -90 ry 0 rz 60 deg; joints []
